  MoveL 667 to (47.33, 219.29, 110) mm, rotated rx -180 ry -65 rz 119.3 deg; joints [-3.014, -1.167, 27.755, -60.199, 92.729, -58.894, -1379.296]
  MoveL 668 to (51.17, 225.17, 120) mm, rotated rx 180 ry -65 rz 125.76 deg; joints [-2.739, -0.589, 26.527, -60.1, 93.267, -59.335, -1385.756]
  MoveL 669 to (54.3, 231.49, 130) mm, rotated rx 180 ry -65 rz 132.3 deg; joints [-2.464, 0.043, 25.187, -60.012, 93.835, -59.826, -1392.295]
  MoveL 670 to (56.65, 238.12, 140) mm, rotated rx -180 ry -65 rz 138.89 deg; joints [-2.19, 0.746, 23.7, -59.937, 94.442, -60.381, -1398.886]
  MoveL 671 to (58.18, 244.95, 150) mm, rotated rx -180 ry -65 rz 145.5 deg; joints [-1.917, 1.551, 22.008, -59.879, 95.103, -61.026, -1405.497]
  MoveL 672 to (58.89, 251.83, 160) mm, rotated rx -180 ry -65 rz 152.1 deg; joints [-1.644, 2.509, 20.004, -59.847, 95.845, -61.808, -1412.098]
  MoveL 673 to (58.8, 258.62, 170) mm, rotated rx -180 ry -65 rz 158.66 deg; joints [-1.372, 3.749, 17.431, -59.859, 96.733, -62.841, -1418.655]
  MoveL 674 to (57.96, 265.2, 180) mm, rotated rx 180 ry -65 rz 165.13 deg; joints [-1.101, 5.868, 13.081, -60.001, 98.071, -64.658, -1425.13]
  MoveL 675 to (55.81, 269.32, 189.23) mm, rotated rx -180 ry -65 rz 171.49 deg; joints [-0.831, 7.347, 10.028, -60.103, 99.08, -65.909, -1431.486]
  MoveL 676 to (53.44, 272.3, 198.22) mm, rotated rx -180 ry -65 rz 177.68 deg; joints [-0.562, 7.315, 10.028, -60.006, 99.318, -65.806, -1437.679]
  MoveL 677 to (51.74, 282.68, 210) mm, rotated rx -180 ry -65 rz 173.67 deg; joints [-0.015, -1.146, 27.158, -56.839, 99.081, -66.843, -1443.668]
  MoveL 678 to (48.8, 287.5, 220) mm, rotated rx -180 ry -65 rz 179.41 deg; joints [0.256, -0.417, 25.625, -56.812, 99.725, -67.39, -1449.406]
  MoveL 679 to (45.62, 291.76, 230) mm, rotated rx -180 ry -65 rz -175.15 deg; joints [0.525, 0.414, 23.888, -56.81, 100.426, -68.024, -1454.846]
  MoveL 680 to (42.34, 295.45, 240) mm, rotated rx -180 ry -65 rz -170.06 deg; joints [0.793, 1.393, 21.855, -56.845, 101.208, -68.785, -1459.941]
  MoveL 681 to (39.07, 298.58, 250) mm, rotated rx 180 ry -65 rz -165.36 deg; joints [1.06, 2.615, 19.337, -56.939, 102.123, -69.757, -1464.643]
  MoveL 682 to (35.92, 301.18, 260) mm, rotated rx -180 ry -65 rz -161.09 deg; joints [1.326, 4.38, 15.722, -57.163, 103.337, -71.21, -1468.905]
  MoveL 683 to (33.57, 302.05, 269.47) mm, rotated rx -180 ry -65 rz -157.32 deg; joints [1.591, 7.175, 10.028, -57.664, 105.11, -73.59, -1472.679]
  MoveL 684 to (32.63, 300.8, 278.13) mm, rotated rx 180 ry -65 rz -154.08 deg; joints [1.855, 7.155, 10.028, -57.554, 105.334, -73.468, -1475.919]
  MoveL 685 to (28.22, 306.19, 290) mm, rotated rx 180 ry -65 rz -161.42 deg; joints [2.42, 15.299, -6.738, -59.336, 114.508, -89.823, -1478.582]
  MoveL 686 to (-21.11, 309.47, 290) mm, rotated rx -180 ry -65 rz -106.89 deg; joints [2.421, 15.322, -6.805, -59.353, 114.532, -89.864, -1533.11]
  Set speed (60.0 mm/s)
  MoveL 687 to (-14.3, 309.76, 278.22) mm, rotated rx 180 ry -65 rz -99.58 deg; joints [1.857, 7.138, 10.028, -57.557, 105.344, -73.482, -1530.424]
  MoveL 688 to (-14.79, 311.04, 269.6) mm, rotated rx -180 ry -65 rz -102.86 deg; joints [1.594, 7.151, 10.028, -57.668, 105.125, -73.61, -1527.138]
  MoveL 689 to (-12.3, 312.09, 260) mm, rotated rx 180 ry -65 rz -106.71 deg; joints [1.33, 4.033, 16.354, -57.105, 103.186, -70.962, -1523.29]
  MoveL 690 to (-8.28, 312.8, 250) mm, rotated rx 180 ry -65 rz -111.08 deg; joints [1.065, 2.314, 19.855, -56.897, 102.008, -69.568, -1518.917]
  MoveL 691 to (-3.78, 313.26, 240) mm, rotated rx -180 ry -65 rz -115.94 deg; joints [0.799, 1.083, 22.369, -56.808, 101.101, -68.608, -1514.059]
  MoveL 692 to (1.16, 313.37, 230) mm, rotated rx 180 ry -65 rz -121.24 deg; joints [0.532, 0.083, 24.421, -56.775, 100.321, -67.848, -1508.756]
  MoveL 693 to (6.46, 313.03, 220) mm, rotated rx -180 ry -65 rz -126.95 deg; joints [0.264, -0.774, 26.185, -56.778, 99.621, -67.213, -1503.053]
  MoveL 694 to (12.04, 312.14, 210) mm, rotated rx -180 ry -65 rz -133.01 deg; joints [-0.005, -1.528, 27.745, -56.807, 98.976, -66.664, -1496.995]
  MoveL 695 to (20.33, 307.92, 198.7) mm, rotated rx -180 ry -65 rz -129.37 deg; joints [-0.551, 7.214, 10.028, -60.017, 99.377, -65.89, -1490.629]
  MoveL 696 to (24.04, 307.87, 189.76) mm, rotated rx -180 ry -65 rz -135.99 deg; joints [-0.82, 7.235, 10.028, -60.114, 99.145, -66.001, -1484.006]
  MoveL 697 to (29.38, 305.54, 180) mm, rotated rx -180 ry -65 rz -142.82 deg; joints [-1.089, 4.255, 16.095, -59.831, 97.379, -63.429, -1477.176]
  MoveL 698 to (34.94, 301.92, 170) mm, rotated rx 180 ry -65 rz -149.81 deg; joints [-1.359, 2.744, 19.201, -59.778, 96.359, -62.169, -1470.188]
  MoveL 699 to (40.17, 297.58, 160) mm, rotated rx 180 ry -65 rz -156.91 deg; joints [-1.631, 1.662, 21.443, -59.79, 95.559, -61.288, -1463.094]
  MoveL 700 to (44.94, 292.58, 150) mm, rotated rx -180 ry -65 rz -164.06 deg; joints [-1.903, 0.787, 23.27, -59.836, 94.864, -60.588, -1455.941]
  MoveL 701 to (49.15, 286.99, 140) mm, rotated rx -180 ry -65 rz -171.23 deg; joints [-2.176, 0.041, 24.838, -59.902, 94.236, -59.999, -1448.774]
  MoveL 702 to (52.68, 280.9, 130) mm, rotated rx -180 ry -65 rz -178.36 deg; joints [-2.45, -0.613, 26.225, -59.984, 93.655, -59.488, -1441.638]
  MoveL 703 to (55.46, 274.42, 120) mm, rotated rx 180 ry -65 rz 174.57 deg; joints [-2.726, -1.199, 27.475, -60.078, 93.108, -59.035, -1434.572]
  MoveL 704 to (55.84, 263.25, 108.59) mm, rotated rx 180 ry -65 rz 177.61 deg; joints [-3.24, 7.248, 10.028, -62.938, 93.374, -58.249, -1427.613]
  MoveL 705 to (57.58, 258.78, 99.33) mm, rotated rx 180 ry -65 rz 170.79 deg; joints [-3.514, 7.28, 10.028, -63.024, 93.127, -58.339, -1420.794]
  MoveL 706 to (58.95, 253.96, 90) mm, rotated rx -180 ry -65 rz 164.15 deg; joints [-3.787, 8.027, 8.582, -63.145, 93.209, -59.081, -1414.147]
  MoveL 707 to (58.51, 247.24, 80) mm, rotated rx 180 ry -65 rz 157.7 deg; joints [-4.062, 10.496, 3.656, -63.366, 94.079, -61.4, -1407.701]
  MoveL 708 to (57.35, 240.79, 70) mm, rotated rx -180 ry -65 rz 151.48 deg; joints [-4.337, 11.761, 1.161, -63.52, 94.39, -62.623, -1401.482]
  MoveL 709 to (55.55, 234.7, 60) mm, rotated rx -180 ry -65 rz 145.52 deg; joints [-4.613, 12.736, -0.752, -63.655, 94.566, -63.585, -1395.517]
  MoveL 710 to (53.21, 229.07, 50) mm, rotated rx -180 ry -65 rz 139.83 deg; joints [-4.889, 13.558, -2.357, -63.777, 94.67, -64.411, -1389.83]
  MoveL 711 to (50.45, 223.94, 40) mm, rotated rx 180 ry -65 rz 134.45 deg; joints [-5.166, 14.279, -3.764, -63.889, 94.728, -65.148, -1384.447]
  MoveL 712 to (47.39, 219.37, 30) mm, rotated rx 180 ry -65 rz 129.39 deg; joints [-5.444, 14.929, -5.029, -63.994, 94.753, -65.823, -1379.391]
  MoveL 713 to (44.15, 215.37, 20) mm, rotated rx 180 ry -65 rz 124.69 deg; joints [-5.721, 15.523, -6.184, -64.093, 94.753, -66.45, -1374.688]
  MoveL 714 to (40.85, 211.93, 10) mm, rotated rx -180 ry -65 rz 120.36 deg; joints [-6, 16.071, -7.253, -64.186, 94.732, -67.04, -1370.363]
  MoveL 715 to (33.26, 208.35, -1.05) mm, rotated rx 180 ry -65 rz 126.44 deg; joints [-6.466, 7.153, 10.028, -66.357, 87.195, -50.6, -1366.442]
  MoveL 716 to (-21.11, 309.47, 290) mm, rotated rx -180 ry -65 rz -106.89 deg; joints [2.421, 15.322, -6.805, -59.353, 114.532, -89.864, -1533.11]
  Set speed (60.0 mm/s)
  MoveL 717 to (-34.79, 325.15, 290) mm, rotated rx -180 ry -65 rz -101.9 deg; joints [2.347, 13.614, -2.112, -58.26, 112.923, -87.117, -1538.101]
  MoveL 718 to (33.26, 208.35, -1.05) mm, rotated rx -180 ry -65 rz 126.44 deg; joints [-6.466, 7.153, 10.028, -66.357, 87.195, -50.6, -1366.442]
  Set speed (60.0 mm/s)
  MoveL 719 to (55.59, 198.58, 0) mm, rotated rx 180 ry -65 rz 122.15 deg; joints [-6.324, 15.031, -3.912, -64.104, 93.441, -65.104, -1372.15]
  MoveL 720 to (33.26, 208.35, -1.05) mm, rotated rx -180 ry -65 rz 126.44 deg; joints [-6.466, 7.153, 10.028, -66.357, 87.195, -50.6, -1366.442]
  Set speed (60.0 mm/s)
  MoveL 721 to (40.85, 211.93, 10) mm, rotated rx -180 ry -65 rz 120.36 deg; joints [-6, 16.071, -7.253, -64.186, 94.732, -67.04, -1370.363]
  MoveL 722 to (44.15, 215.37, 20) mm, rotated rx 180 ry -65 rz 124.69 deg; joints [-5.721, 15.523, -6.184, -64.093, 94.753, -66.45, -1374.688]
  MoveL 723 to (47.39, 219.37, 30) mm, rotated rx 180 ry -65 rz 129.39 deg; joints [-5.444, 14.929, -5.029, -63.994, 94.753, -65.823, -1379.391]
  MoveL 724 to (50.45, 223.94, 40) mm, rotated rx 180 ry -65 rz 134.45 deg; joints [-5.166, 14.279, -3.764, -63.889, 94.728, -65.148, -1384.447]
  MoveL 725 to (53.21, 229.07, 50) mm, rotated rx -180 ry -65 rz 139.83 deg; joints [-4.889, 13.558, -2.357, -63.777, 94.67, -64.411, -1389.83]
  MoveL 726 to (55.55, 234.7, 60) mm, rotated rx 180 ry -65 rz 145.52 deg; joints [-4.613, 12.736, -0.752, -63.655, 94.566, -63.585, -1395.517]
  MoveL 727 to (57.35, 240.79, 70) mm, rotated rx -180 ry -65 rz 151.48 deg; joints [-4.337, 11.761, 1.161, -63.52, 94.39, -62.623, -1401.482]
  MoveL 728 to (58.51, 247.24, 80) mm, rotated rx 180 ry -65 rz 157.7 deg; joints [-4.062, 10.496, 3.656, -63.366, 94.079, -61.4, -1407.701]
  MoveL 729 to (58.95, 253.96, 90) mm, rotated rx 180 ry -65 rz 164.15 deg; joints [-3.787, 8.027, 8.582, -63.145, 93.209, -59.081, -1414.147]
  MoveL 730 to (57.58, 258.78, 99.33) mm, rotated rx -180 ry -65 rz 170.79 deg; joints [-3.514, 7.28, 10.028, -63.024, 93.127, -58.339, -1420.794]
  MoveL 731 to (55.84, 263.25, 108.59) mm, rotated rx 180 ry -65 rz 177.61 deg; joints [-3.24, 7.248, 10.028, -62.938, 93.374, -58.249, -1427.613]
  MoveL 732 to (55.46, 274.42, 120) mm, rotated rx -180 ry -65 rz 174.57 deg; joints [-2.726, 16.068, -7.419, -62.097, 101.684, -74.582, -1434.572]
  MoveL 733 to (52.68, 280.9, 130) mm, rotated rx 180 ry -65 rz -178.36 deg; joints [-2.45, 15.417, -6.169, -61.918, 101.643, -73.911, -1441.638]
  MoveL 734 to (49.15, 286.99, 140) mm, rotated rx -180 ry -65 rz -171.23 deg; joints [-2.176, 14.699, -4.782, -61.726, 101.566, -73.179, -1448.774]
  MoveL 735 to (44.94, 292.58, 150) mm, rotated rx -180 ry -65 rz -164.06 deg; joints [-1.903, 13.892, -3.214, -61.514, 101.44, -72.365, -1455.941]
  MoveL 736 to (40.17, 297.58, 160) mm, rotated rx -180 ry -65 rz -156.91 deg; joints [-1.631, 12.959, -1.387, -61.279, 101.247, -71.434, -1463.094]
  MoveL 737 to (34.94, 301.92, 170) mm, rotated rx -180 ry -65 rz -149.81 deg; joints [-1.359, 11.822, 0.855, -61.007, 100.945, -70.317, -1470.188]
  MoveL 738 to (29.38, 305.54, 180) mm, rotated rx -180 ry -65 rz -142.82 deg; joints [-1.089, 10.261, 3.96, -60.665, 100.423, -68.815, -1477.176]
  MoveL 739 to (24.04, 307.87, 189.76) mm, rotated rx 180 ry -65 rz -135.99 deg; joints [-0.82, 7.235, 10.028, -60.114, 99.145, -66.001, -1484.006]
  MoveL 740 to (20.33, 307.92, 198.7) mm, rotated rx -180 ry -65 rz -129.37 deg; joints [-0.551, 7.214, 10.028, -60.017, 99.377, -65.89, -1490.629]
  MoveL 741 to (12.04, 312.14, 210) mm, rotated rx 180 ry -65 rz -133.01 deg; joints [-0.005, -1.528, 27.745, -56.807, 98.976, -66.664, -1496.995]
  MoveL 742 to (6.46, 313.03, 220) mm, rotated rx 180 ry -65 rz -126.95 deg; joints [0.264, -0.774, 26.185, -56.778, 99.621, -67.213, -1503.053]
  MoveL 743 to (1.16, 313.37, 230) mm, rotated rx 180 ry -65 rz -121.24 deg; joints [0.532, 0.083, 24.421, -56.775, 100.321, -67.848, -1508.756]
  MoveL 744 to (-3.78, 313.26, 240) mm, rotated rx 180 ry -65 rz -115.94 deg; joints [0.799, 1.083, 22.369, -56.808, 101.101, -68.608, -1514.059]
  MoveL 745 to (-8.28, 312.8, 250) mm, rotated rx -180 ry -65 rz -111.08 deg; joints [1.065, 2.314, 19.855, -56.897, 102.008, -69.568, -1518.917]
  MoveL 746 to (-12.3, 312.09, 260) mm, rotated rx 180 ry -65 rz -106.71 deg; joints [1.33, 4.033, 16.354, -57.105, 103.186, -70.962, -1523.29]
  MoveL 747 to (-14.79, 311.04, 269.6) mm, rotated rx -180 ry -65 rz -102.86 deg; joints [1.594, 7.151, 10.028, -57.668, 105.125, -73.61, -1527.138]
  MoveL 748 to (-14.3, 309.76, 278.22) mm, rotated rx -180 ry -65 rz -99.58 deg; joints [1.857, 7.138, 10.028, -57.557, 105.344, -73.482, -1530.424]
  MoveL 749 to (-21.11, 309.47, 290) mm, rotated rx 180 ry -65 rz -106.89 deg; joints [2.421, -1.338, 26.861, -54.18, 105.153, -74.752, -1533.11]
  MoveL 750 to (-34.79, 325.15, 290) mm, rotated rx -180 ry -65 rz -101.9 deg; joints [2.347, 1.599, 22.168, -54.622, 106.121, -76.277, -1538.101]
  Set speed (60.0 mm/s)
  MoveL 751 to (-31.73, 326.57, 280) mm, rotated rx -180 ry -65 rz -104.51 deg; joints [2.083, 0.505, 24.407, -54.508, 105.261, -75.453, -1535.486]
  MoveL 752 to (-27.92, 328.13, 270) mm, rotated rx 180 ry -65 rz -107.71 deg; joints [1.818, -0.43, 26.324, -54.446, 104.496, -74.77, -1532.288]
  MoveL 753 to (-17.68, 328.71, 257.77) mm, rotated rx 180 ry -65 rz -101.46 deg; joints [1.26, 7.769, 10.028, -57.675, 104.526, -73.246, -1528.542]
  MoveL 754 to (-15.78, 330.54, 249.09) mm, rotated rx -180 ry -65 rz -105.71 deg; joints [0.996, 7.782, 10.028, -57.788, 104.306, -73.373, -1524.286]
  MoveL 755 to (-12.17, 332.29, 240) mm, rotated rx -180 ry -65 rz -110.44 deg; joints [0.731, 5.846, 13.967, -57.494, 103.022, -71.769, -1519.557]
  MoveL 756 to (-5.61, 333.04, 230) mm, rotated rx -180 ry -65 rz -115.61 deg; joints [0.465, 3.66, 18.415, -57.203, 101.592, -69.958, -1514.392]
  MoveL 757 to (1.49, 333.22, 220) mm, rotated rx -180 ry -65 rz -121.17 deg; joints [0.198, 2.31, 21.174, -57.1, 100.621, -68.887, -1508.834]
  MoveL 758 to (9.03, 332.72, 210) mm, rotated rx -180 ry -65 rz -127.08 deg; joints [-0.071, 1.257, 23.337, -57.066, 99.812, -68.076, -1502.922]
  MoveL 759 to (16.88, 331.41, 200) mm, rotated rx -180 ry -65 rz -133.3 deg; joints [-0.34, 0.375, 25.158, -57.071, 99.097, -67.411, -1496.702]
  MoveL 760 to (24.89, 329.2, 190) mm, rotated rx -180 ry -65 rz -139.78 deg; joints [-0.61, -0.391, 26.749, -57.103, 98.444, -66.845, -1490.217]
  MoveL 761 to (36.37, 321.13, 177.97) mm, rotated rx 180 ry -65 rz -136.49 deg; joints [-1.15, 7.85, 10.028, -60.155, 98.565, -65.62, -1483.513]
  MoveL 762 to (42.24, 319.12, 168.96) mm, rotated rx -180 ry -65 rz -143.36 deg; joints [-1.42, 7.875, 10.028, -60.254, 98.331, -65.728, -1476.637]
  MoveL 763 to (48.36, 316.44, 159.89) mm, rotated rx -180 ry -65 rz -150.37 deg; joints [-1.69, 7.901, 10.028, -60.352, 98.094, -65.833, -1469.635]
  MoveL 764 to (55.2, 310.67, 150) mm, rotated rx 180 ry -65 rz -157.45 deg; joints [-1.962, 11.044, 3.733, -60.871, 99.414, -68.741, -1462.551]
  MoveL 765 to (61.48, 303.74, 140) mm, rotated rx -180 ry -65 rz -164.57 deg; joints [-2.234, 12.483, 0.887, -61.168, 99.865, -70.12, -1455.431]
  MoveL 766 to (66.92, 296.06, 130) mm, rotated rx -180 ry -65 rz -171.68 deg; joints [-2.507, 13.555, -1.216, -61.411, 100.126, -71.168, -1448.317]
  MoveL 767 to (71.41, 287.77, 120) mm, rotated rx 180 ry -65 rz -178.75 deg; joints [-2.782, 14.443, -2.946, -61.624, 100.292, -72.05, -1441.249]
  MoveL 768 to (74.87, 279.04, 110) mm, rotated rx -180 ry -65 rz 174.27 deg; joints [-3.057, 15.216, -4.44, -61.816, 100.396, -72.826, -1434.266]
  MoveL 769 to (77.24, 270.04, 100) mm, rotated rx -180 ry -65 rz 167.4 deg; joints [-3.333, 15.907, -5.769, -61.993, 100.457, -73.527, -1427.404]
  MoveL 770 to (78.53, 260.95, 90) mm, rotated rx 180 ry -65 rz 160.7 deg; joints [-3.609, 16.536, -6.973, -62.158, 100.485, -74.174, -1420.696]
  MoveL 771 to (75.48, 247.1, 78.35) mm, rotated rx -180 ry -65 rz 164.17 deg; joints [-4.113, 7.925, 10.028, -63.191, 92.325, -58.021, -1414.174]
  MoveL 772 to (75.7, 240.53, 69.02) mm, rotated rx 180 ry -65 rz 157.87 deg; joints [-4.388, 7.956, 10.028, -63.279, 92.078, -58.111, -1407.868]
  MoveL 773 to (75.43, 234.04, 59.66) mm, rotated rx -180 ry -65 rz 151.81 deg; joints [-4.663, 7.986, 10.028, -63.367, 91.831, -58.202, -1401.808]
  MoveL 774 to (73.92, 227.12, 50) mm, rotated rx -180 ry -65 rz 146.02 deg; joints [-4.938, 6.02, 14.06, -63.419, 90.673, -56.471, -1396.021]
  MoveL 775 to (70.87, 219.96, 40) mm, rotated rx -180 ry -65 rz 140.54 deg; joints [-5.214, 4.454, 17.278, -63.513, 89.704, -55.108, -1390.535]
  MoveL 776 to (67.34, 213.5, 30) mm, rotated rx 180 ry -65 rz 135.38 deg; joints [-5.491, 3.412, 19.436, -63.628, 88.978, -54.223, -1385.378]
  MoveL 777 to (63.51, 207.78, 20) mm, rotated rx -180 ry -65 rz 130.58 deg; joints [-5.768, 2.578, 21.169, -63.754, 88.351, -53.53, -1380.576]
  MoveL 778 to (59.54, 202.81, 10) mm, rotated rx -180 ry -65 rz 126.16 deg; joints [-6.046, 1.865, 22.654, -63.887, 87.783, -52.949, -1376.157]
  MoveL 779 to (55.59, 198.58, 0) mm, rotated rx -180 ry -65 rz 122.15 deg; joints [-6.324, 1.235, 23.968, -64.026, 87.256, -52.444, -1372.15]
  MoveL 780 to (-34.79, 325.15, 290) mm, rotated rx 180 ry -65 rz -101.9 deg; joints [2.347, 1.599, 22.168, -54.622, 106.121, -76.277, -1538.101]
  Set speed (60.0 mm/s)
  MoveL 781 to (-30.72, 304.75, 290) mm, rotated rx 180 ry -65 rz -95.53 deg; joints [2.42, -1.275, 26.764, -54.188, 105.172, -74.782, -1544.467]
  MoveL 782 to (55.59, 198.58, 0) mm, rotated rx 180 ry -65 rz 122.15 deg; joints [-6.324, 1.235, 23.968, -64.026, 87.256, -52.444, -1372.15]
  Set speed (60.0 mm/s)
  MoveL 783 to (41.3, 215.27, -0.99) mm, rotated rx 180 ry -65 rz 136.17 deg; joints [-6.465, 7.133, 10.028, -66.356, 87.204, -50.617, -1376.169]
  MoveL 784 to (55.59, 198.58, 0) mm, rotated rx -180 ry -65 rz 122.15 deg; joints [-6.324, 1.235, 23.968, -64.026, 87.256, -52.444, -1372.15]
  Set speed (60.0 mm/s)
  MoveL 785 to (59.54, 202.81, 10) mm, rotated rx -180 ry -65 rz 126.16 deg; joints [-6.046, 1.865, 22.654, -63.887, 87.783, -52.949, -1376.157]
  MoveL 786 to (63.51, 207.78, 20) mm, rotated rx -180 ry -65 rz 130.58 deg; joints [-5.768, 2.578, 21.169, -63.754, 88.351, -53.53, -1380.576]
  MoveL 787 to (67.34, 213.5, 30) mm, rotated rx -180 ry -65 rz 135.38 deg; joints [-5.491, 3.412, 19.436, -63.628, 88.978, -54.223, -1385.378]
  MoveL 788 to (70.87, 219.96, 40) mm, rotated rx 180 ry -65 rz 140.54 deg; joints [-5.214, 4.454, 17.278, -63.513, 89.704, -55.108, -1390.535]
  MoveL 789 to (73.92, 227.12, 50) mm, rotated rx 180 ry -65 rz 146.02 deg; joints [-4.938, 6.02, 14.06, -63.419, 90.673, -56.471, -1396.021]
  MoveL 790 to (75.43, 234.04, 59.66) mm, rotated rx -180 ry -65 rz 151.81 deg; joints [-4.663, 7.986, 10.028, -63.367, 91.831, -58.202, -1401.808]
  MoveL 791 to (75.7, 240.53, 69.02) mm, rotated rx -180 ry -65 rz 157.87 deg; joints [-4.388, 7.956, 10.028, -63.279, 92.078, -58.111, -1407.868]
  MoveL 792 to (75.48, 247.1, 78.35) mm, rotated rx 180 ry -65 rz 164.17 deg; joints [-4.113, 7.925, 10.028, -63.191, 92.325, -58.021, -1414.174]
  MoveL 793 to (78.53, 260.95, 90) mm, rotated rx -180 ry -65 rz 160.7 deg; joints [-3.609, -0.289, 27.028, -60.472, 92.192, -59.025, -1420.696]
  MoveL 794 to (77.24, 270.04, 100) mm, rotated rx 180 ry -65 rz 167.4 deg; joints [-3.333, 0.273, 25.825, -60.367, 92.724, -59.461, -1427.404]
  MoveL 795 to (74.87, 279.04, 110) mm, rotated rx -180 ry -65 rz 174.27 deg; joints [-3.057, 0.897, 24.496, -60.273, 93.289, -59.951, -1434.266]
  MoveL 796 to (71.41, 287.77, 120) mm, rotated rx -180 ry -65 rz -178.75 deg; joints [-2.782, 1.603, 23.002, -60.192, 93.897, -60.513, -1441.249]
  MoveL 797 to (66.92, 296.06, 130) mm, rotated rx -180 ry -65 rz -171.68 deg; joints [-2.507, 2.427, 21.272, -60.129, 94.565, -61.176, -1448.317]
  MoveL 798 to (61.48, 303.74, 140) mm, rotated rx 180 ry -65 rz -164.57 deg; joints [-2.234, 3.436, 19.169, -60.093, 95.328, -62.003, -1455.431]
  MoveL 799 to (55.2, 310.67, 150) mm, rotated rx -180 ry -65 rz -157.45 deg; joints [-1.962, 4.814, 16.322, -60.108, 96.279, -63.155, -1462.551]
  MoveL 800 to (48.36, 316.44, 159.89) mm, rotated rx 180 ry -65 rz -150.37 deg; joints [-1.69, 7.901, 10.028, -60.352, 98.094, -65.833, -1469.635]
  MoveL 801 to (42.24, 319.12, 168.96) mm, rotated rx -180 ry -65 rz -143.36 deg; joints [-1.42, 7.875, 10.028, -60.254, 98.331, -65.728, -1476.637]
  MoveL 802 to (36.37, 321.13, 177.97) mm, rotated rx -180 ry -65 rz -136.49 deg; joints [-1.15, 7.85, 10.028, -60.155, 98.565, -65.62, -1483.513]
  MoveL 803 to (24.89, 329.2, 190) mm, rotated rx -180 ry -65 rz -139.78 deg; joints [-0.61, 16.157, -6.693, -60.422, 107.256, -81.648, -1490.217]
  MoveL 804 to (16.88, 331.41, 200) mm, rotated rx 180 ry -65 rz -133.3 deg; joints [-0.34, 15.349, -5.102, -60.125, 107.099, -80.798, -1496.702]
  MoveL 805 to (9.03, 332.72, 210) mm, rotated rx -180 ry -65 rz -127.08 deg; joints [-0.071, 14.429, -3.281, -59.796, 106.877, -79.844, -1502.922]
  MoveL 806 to (1.49, 333.22, 220) mm, rotated rx 180 ry -65 rz -121.17 deg; joints [0.198, 13.342, -1.118, -59.423, 106.559, -78.736, -1508.834]
  MoveL 807 to (-5.61, 333.04, 230) mm, rotated rx -180 ry -65 rz -115.61 deg; joints [0.465, 11.961, 1.641, -58.978, 106.077, -77.364, -1514.392]
  MoveL 808 to (-12.17, 332.29, 240) mm, rotated rx -180 ry -65 rz -110.44 deg; joints [0.731, 9.745, 6.088, -58.34, 105.136, -75.246, -1519.557]
  MoveL 809 to (-15.78, 330.54, 249.09) mm, rotated rx -180 ry -65 rz -105.71 deg; joints [0.996, 7.782, 10.028, -57.788, 104.306, -73.373, -1524.286]
  MoveL 810 to (-17.68, 328.71, 257.77) mm, rotated rx -180 ry -65 rz -101.46 deg; joints [1.26, 7.769, 10.028, -57.675, 104.526, -73.246, -1528.542]
  MoveL 811 to (-27.92, 328.13, 270) mm, rotated rx 180 ry -65 rz -107.71 deg; joints [1.818, 15.697, -6.268, -59.233, 113.553, -89.338, -1532.288]
  MoveL 812 to (-31.73, 326.57, 280) mm, rotated rx -180 ry -65 rz -104.51 deg; joints [2.083, 14.735, -4.351, -58.774, 113.285, -88.299, -1535.486]
  MoveL 813 to (-34.79, 325.15, 290) mm, rotated rx -180 ry -65 rz -101.9 deg; joints [2.347, 13.614, -2.112, -58.26, 112.923, -87.117, -1538.101]
  MoveL 814 to (-30.72, 304.75, 290) mm, rotated rx 180 ry -65 rz -95.53 deg; joints [2.42, 15.288, -6.708, -59.329, 114.498, -89.805, -1544.467]
  Set speed (60.0 mm/s)
  MoveL 815 to (-23.89, 306.35, 278.15) mm, rotated rx 180 ry -65 rz -88.19 deg; joints [1.855, 7.151, 10.028, -57.554, 105.336, -73.471, -1541.806]
  MoveL 816 to (-24.62, 307.45, 269.53) mm, rotated rx -180 ry -65 rz -91.45 deg; joints [1.592, 7.162, 10.028, -57.666, 105.118, -73.6, -1538.548]
  MoveL 817 to (-22.53, 308.91, 260) mm, rotated rx -180 ry -65 rz -95.27 deg; joints [1.329, 10.215, 3.881, -58.52, 106.538, -76.47, -1534.728]
  MoveL 818 to (-18.7, 310.34, 250) mm, rotated rx -180 ry -65 rz -99.62 deg; joints [1.064, 12.003, 0.29, -59.089, 107.252, -78.221, -1530.381]
  MoveL 819 to (-14.35, 311.61, 240) mm, rotated rx 180 ry -65 rz -104.46 deg; joints [0.799, 13.279, -2.266, -59.531, 107.681, -79.514, -1525.543]
  MoveL 820 to (-9.52, 312.61, 230) mm, rotated rx -180 ry -65 rz -109.75 deg; joints [0.532, 14.321, -4.347, -59.911, 107.979, -80.596, -1520.254]
  MoveL 821 to (-4.24, 313.23, 220) mm, rotated rx 180 ry -65 rz -115.45 deg; joints [0.265, 15.218, -6.134, -60.25, 108.194, -81.546, -1514.554]
  MoveL 822 to (1.41, 313.37, 210) mm, rotated rx 180 ry -65 rz -121.51 deg; joints [-0.004, 16.014, -7.714, -60.559, 108.35, -82.402, -1508.487]
  MoveL 823 to (10.28, 310.83, 198.74) mm, rotated rx -180 ry -65 rz -117.9 deg; joints [-0.551, 7.207, 10.028, -60.017, 99.382, -65.896, -1502.098]
  MoveL 824 to (13.88, 311.45, 189.81) mm, rotated rx -180 ry -65 rz -124.57 deg; joints [-0.818, 7.224, 10.028, -60.115, 99.151, -66.01, -1495.435]
  MoveL 825 to (19.65, 310.01, 180) mm, rotated rx -180 ry -65 rz -131.45 deg; joints [-1.087, 4.115, 16.351, -59.818, 97.322, -63.328, -1488.548]
  MoveL 826 to (25.78, 307.45, 170) mm, rotated rx 180 ry -65 rz -138.51 deg; joints [-1.357, 2.623, 19.411, -59.769, 96.316, -62.091, -1481.489]
  MoveL 827 to (31.7, 304.13, 160) mm, rotated rx 180 ry -65 rz -145.69 deg; joints [-1.628, 1.542, 21.643, -59.783, 95.52, -61.217, -1474.307]
  MoveL 828 to (37.3, 300.08, 150) mm, rotated rx -180 ry -65 rz -152.95 deg; joints [-1.901, 0.666, 23.467, -59.829, 94.828, -60.521, -1467.054]
  MoveL 829 to (42.45, 295.34, 140) mm, rotated rx 180 ry -65 rz -160.22 deg; joints [-2.174, -0.08, 25.033, -59.896, 94.202, -59.935, -1459.778]
  MoveL 830 to (47.02, 289.99, 130) mm, rotated rx 180 ry -65 rz -167.48 deg; joints [-2.448, -0.735, 26.417, -59.979, 93.622, -59.427, -1452.524]
  MoveL 831 to (50.93, 284.12, 120) mm, rotated rx -180 ry -65 rz -174.66 deg; joints [-2.723, -1.321, 27.664, -60.073, 93.077, -58.977, -1445.337]
  MoveL 832 to (53.41, 273.61, 108.72) mm, rotated rx -180 ry -65 rz -171.74 deg; joints [-3.238, 7.218, 10.028, -62.939, 93.39, -58.274, -1438.256]
  MoveL 833 to (55.97, 269.53, 99.46) mm, rotated rx -180 ry -65 rz -178.68 deg; joints [-3.511, 7.25, 10.028, -63.025, 93.143, -58.365, -1431.316]
  MoveL 834 to (58.06, 264.62, 90) mm, rotated rx -180 ry -65 rz 174.55 deg; joints [-3.785, 8.775, 7.009, -63.188, 93.584, -59.818, -1424.553]
  MoveL 835 to (58.85, 257.94, 80) mm, rotated rx 180 ry -65 rz 168 deg; joints [-4.059, 10.726, 3.129, -63.384, 94.214, -61.664, -1417.997]
  MoveL 836 to (58.87, 251.39, 70) mm, rotated rx -180 ry -65 rz 161.68 deg; joints [-4.335, 11.918, 0.782, -63.535, 94.491, -62.821, -1411.675]
  MoveL 837 to (58.2, 245.07, 60) mm, rotated rx -180 ry -65 rz 155.62 deg; joints [-4.61, 12.858, -1.057, -63.668, 94.649, -63.749, -1405.616]
  MoveL 838 to (56.92, 239.11, 50) mm, rotated rx 180 ry -65 rz 149.84 deg; joints [-4.887, 13.657, -2.614, -63.788, 94.742, -64.551, -1399.845]
  MoveL 839 to (55.13, 233.57, 40) mm, rotated rx 180 ry -65 rz 144.39 deg; joints [-5.164, 14.362, -3.984, -63.899, 94.791, -65.271, -1394.385]
  MoveL 840 to (52.95, 228.52, 30) mm, rotated rx -180 ry -65 rz 139.26 deg; joints [-5.442, 14.998, -5.22, -64.003, 94.808, -65.932, -1389.263]
  MoveL 841 to (50.48, 223.99, 20) mm, rotated rx 180 ry -65 rz 134.5 deg; joints [-5.72, 15.582, -6.351, -64.101, 94.802, -66.547, -1384.503]
  MoveL 842 to (42.09, 217.59, 8.47) mm, rotated rx -180 ry -65 rz 140.13 deg; joints [-6.189, 7.114, 10.028, -66.279, 87.453, -50.529, -1380.13]
  MoveL 843 to (41.3, 215.27, -0.99) mm, rotated rx 180 ry -65 rz 136.17 deg; joints [-6.465, 7.133, 10.028, -66.356, 87.204, -50.617, -1376.169]
  MoveL 844 to (-30.72, 304.75, 290) mm, rotated rx -180 ry -65 rz -95.53 deg; joints [2.42, 15.288, -6.708, -59.329, 114.498, -89.805, -1544.467]
  Set speed (60.0 mm/s)
  MoveL 845 to (-58.22, 263.67, 290) mm, rotated rx -180 ry -65 rz -43.61 deg; joints [2.405, 14.999, -5.871, -59.121, 114.205, -89.297, -1596.394]
  MoveL 846 to (41.3, 215.27, -0.99) mm, rotated rx 180 ry -65 rz 136.17 deg; joints [-6.465, 7.133, 10.028, -66.356, 87.204, -50.617, -1736.169]
  Set speed (60.0 mm/s)
  MoveL 847 to (57.25, 262.28, -0.53) mm, rotated rx -180 ry -65 rz -175.75 deg; joints [-6.455, 7, 10.028, -66.348, 87.266, -50.736, -1784.254]
  MoveL 848 to (41.3, 215.27, -0.99) mm, rotated rx -180 ry -65 rz 136.17 deg; joints [-6.465, 7.133, 10.028, -66.356, 87.204, -50.617, -1736.169]
  Set speed (60.0 mm/s)
  MoveL 849 to (42.09, 217.59, 8.47) mm, rotated rx -180 ry -65 rz 140.13 deg; joints [-6.189, 7.114, 10.028, -66.279, 87.453, -50.529, -1740.13]
  MoveL 850 to (50.48, 223.99, 20) mm, rotated rx -180 ry -65 rz 134.5 deg; joints [-5.72, -0.628, 26.407, -63.801, 87.493, -51.686, -1744.503]
  MoveL 851 to (52.95, 228.52, 30) mm, rotated rx 180 ry -65 rz 139.26 deg; joints [-5.442, -0.092, 25.275, -63.664, 87.982, -52.109, -1749.263]
  MoveL 852 to (55.13, 233.57, 40) mm, rotated rx -180 ry -65 rz 144.39 deg; joints [-5.164, 0.494, 24.04, -63.533, 88.496, -52.579, -1754.385]
  MoveL 853 to (56.92, 239.11, 50) mm, rotated rx -180 ry -65 rz 149.84 deg; joints [-4.887, 1.145, 22.67, -63.408, 89.044, -53.11, -1759.845]
  MoveL 854 to (58.2, 245.07, 60) mm, rotated rx -180 ry -65 rz 155.62 deg; joints [-4.61, 1.887, 21.113, -63.291, 89.636, -53.725, -1765.616]
  MoveL 855 to (58.87, 251.39, 70) mm, rotated rx 180 ry -65 rz 161.68 deg; joints [-4.335, 2.768, 19.274, -63.185, 90.295, -54.466, -1771.675]
  MoveL 856 to (58.85, 257.94, 80) mm, rotated rx -180 ry -65 rz 168 deg; joints [-4.059, 3.899, 16.926, -63.096, 91.073, -55.435, -1777.997]
  MoveL 857 to (58.06, 264.62, 90) mm, rotated rx 180 ry -65 rz 174.55 deg; joints [-3.785, 5.787, 13.046, -63.051, 92.205, -57.094, -1784.553]
  MoveL 858 to (55.97, 269.53, 99.46) mm, rotated rx 180 ry -65 rz -178.68 deg; joints [-3.511, 7.25, 10.028, -63.025, 93.143, -58.365, -1791.316]
  MoveL 859 to (53.41, 273.61, 108.72) mm, rotated rx -180 ry -65 rz -171.74 deg; joints [-3.238, 7.218, 10.028, -62.939, 93.39, -58.274, -1798.256]
  MoveL 860 to (50.93, 284.12, 120) mm, rotated rx -180 ry -65 rz -174.66 deg; joints [-2.723, 16.132, -7.608, -62.119, 101.745, -74.693, -1805.337]
  MoveL 861 to (47.02, 289.99, 130) mm, rotated rx 180 ry -65 rz -167.48 deg; joints [-2.448, 15.484, -6.361, -61.941, 101.704, -74.022, -1812.524]
  MoveL 862 to (42.45, 295.34, 140) mm, rotated rx 180 ry -65 rz -160.22 deg; joints [-2.174, 14.769, -4.977, -61.747, 101.626, -73.289, -1819.778]
  MoveL 863 to (37.3, 300.08, 150) mm, rotated rx -180 ry -65 rz -152.95 deg; joints [-1.901, 13.966, -3.411, -61.535, 101.5, -72.474, -1827.054]
  MoveL 864 to (31.7, 304.13, 160) mm, rotated rx 180 ry -65 rz -145.69 deg; joints [-1.628, 13.038, -1.587, -61.299, 101.307, -71.542, -1834.307]
  MoveL 865 to (25.78, 307.45, 170) mm, rotated rx 180 ry -65 rz -138.51 deg; joints [-1.357, 11.909, 0.645, -61.027, 101.007, -70.426, -1841.489]
  MoveL 866 to (19.65, 310.01, 180) mm, rotated rx 180 ry -65 rz -131.45 deg; joints [-1.087, 10.373, 3.705, -60.688, 100.494, -68.941, -1848.548]
  MoveL 867 to (13.88, 311.45, 189.81) mm, rotated rx -180 ry -65 rz -124.57 deg; joints [-0.818, 7.224, 10.028, -60.115, 99.151, -66.01, -1855.435]
  MoveL 868 to (10.28, 310.83, 198.74) mm, rotated rx 180 ry -65 rz -117.9 deg; joints [-0.551, 7.207, 10.028, -60.017, 99.382, -65.896, -1862.098]
  MoveL 869 to (1.41, 313.37, 210) mm, rotated rx -180 ry -65 rz -121.51 deg; joints [-0.004, -1.544, 27.77, -56.806, 98.972, -66.657, -1868.487]
  MoveL 870 to (-4.24, 313.23, 220) mm, rotated rx -180 ry -65 rz -115.45 deg; joints [0.265, -0.777, 26.19, -56.778, 99.62, -67.212, -1874.554]
  MoveL 871 to (-9.52, 312.61, 230) mm, rotated rx 180 ry -65 rz -109.75 deg; joints [0.532, 0.094, 24.402, -56.777, 100.325, -67.855, -1880.254]
  MoveL 872 to (-14.35, 311.61, 240) mm, rotated rx -180 ry -65 rz -104.46 deg; joints [0.799, 1.112, 22.322, -56.811, 101.111, -68.624, -1885.543]
  MoveL 873 to (-18.7, 310.34, 250) mm, rotated rx -180 ry -65 rz -99.62 deg; joints [1.064, 2.365, 19.766, -56.904, 102.028, -69.601, -1890.381]
  MoveL 874 to (-22.53, 308.91, 260) mm, rotated rx -180 ry -65 rz -95.27 deg; joints [1.329, 4.131, 16.175, -57.122, 103.228, -71.032, -1894.728]
  MoveL 875 to (-24.62, 307.45, 269.53) mm, rotated rx 180 ry -65 rz -91.45 deg; joints [1.592, 7.162, 10.028, -57.666, 105.118, -73.6, -1898.548]
  MoveL 876 to (-23.89, 306.35, 278.15) mm, rotated rx 180 ry -65 rz -88.19 deg; joints [1.855, 7.151, 10.028, -57.554, 105.336, -73.471, -1901.806]
  MoveL 877 to (-30.72, 304.75, 290) mm, rotated rx -180 ry -65 rz -95.53 deg; joints [2.42, -1.275, 26.764, -54.188, 105.172, -74.782, -1904.467]
  MoveL 878 to (-58.22, 263.67, 290) mm, rotated rx -180 ry -65 rz -43.61 deg; joints [2.405, -0.736, 25.927, -54.263, 105.335, -75.041, -1956.394]
  Set speed (60.0 mm/s)
  MoveL 879 to (-57.77, 266.15, 280) mm, rotated rx -180 ry -65 rz -46.08 deg; joints [2.141, -1.618, 27.728, -54.215, 104.605, -74.413, -1953.924]
  MoveL 880 to (-55.45, 271.33, 268.93) mm, rotated rx 180 ry -65 rz -39.11 deg; joints [1.579, 7.278, 10.028, -57.645, 105.045, -73.506, -1950.894]
  MoveL 881 to (-56.08, 272.6, 260) mm, rotated rx -180 ry -65 rz -42.67 deg; joints [1.316, 5.488, 13.657, -57.363, 103.847, -72.043, -1947.333]
  MoveL 882 to (-54.69, 276.44, 250) mm, rotated rx -180 ry -65 rz -46.73 deg; joints [1.052, 3.098, 18.494, -57.008, 102.312, -70.069, -1943.267]
  MoveL 883 to (-52.84, 280.57, 240) mm, rotated rx 180 ry -65 rz -51.28 deg; joints [0.788, 1.654, 21.421, -56.876, 101.299, -68.937, -1938.724]
  MoveL 884 to (-50.46, 284.91, 230) mm, rotated rx 180 ry -65 rz -56.27 deg; joints [0.523, 0.519, 23.719, -56.821, 100.459, -68.08, -1933.731]
  MoveL 885 to (-47.51, 289.33, 220) mm, rotated rx -180 ry -65 rz -61.68 deg; joints [0.256, -0.443, 25.665, -56.81, 99.718, -67.377, -1928.316]
  MoveL 886 to (-43.95, 293.72, 210) mm, rotated rx 180 ry -65 rz -67.49 deg; joints [-0.011, -1.288, 27.377, -56.827, 99.042, -66.776, -1922.509]
  MoveL 887 to (-35.74, 299.31, 198.51) mm, rotated rx -180 ry -65 rz -63.66 deg; joints [-0.556, 7.253, 10.028, -60.012, 99.354, -65.858, -1916.342]
  MoveL 888 to (-34, 302.1, 189.66) mm, rotated rx -180 ry -65 rz -70.15 deg; joints [-0.822, 7.255, 10.028, -60.112, 99.133, -65.984, -1909.847]
  MoveL 889 to (-29.57, 305.43, 180) mm, rotated rx -180 ry -65 rz -76.94 deg; joints [-1.089, 10.258, 3.967, -60.665, 100.421, -68.812, -1903.063]
  MoveL 890 to (-23.65, 308.43, 170) mm, rotated rx 180 ry -65 rz -83.97 deg; joints [-1.357, 11.924, 0.608, -61.031, 101.018, -70.445, -1896.03]
  MoveL 891 to (-17.28, 310.79, 160) mm, rotated rx 180 ry -65 rz -91.21 deg; joints [-1.626, 13.117, -1.789, -61.32, 101.368, -71.651, -1888.791]
  MoveL 892 to (-10.57, 312.43, 150) mm, rotated rx 180 ry -65 rz -98.61 deg; joints [-1.897, 14.087, -3.734, -61.571, 101.6, -72.653, -1881.395]
  MoveL 893 to (-3.62, 313.27, 140) mm, rotated rx 180 ry -65 rz -106.11 deg; joints [-2.168, 14.92, -5.395, -61.795, 101.758, -73.528, -1873.889]
  MoveL 894 to (3.42, 313.28, 130) mm, rotated rx -180 ry -65 rz -113.67 deg; joints [-2.441, 15.657, -6.857, -61.998, 101.862, -74.311, -1866.327]
  MoveL 895 to (14.77, 308.97, 118.31) mm, rotated rx -180 ry -65 rz -111.24 deg; joints [-2.957, 7.1, 10.028, -62.855, 93.682, -58.257, -1858.761]
  MoveL 896 to (19.25, 308.72, 109.14) mm, rotated rx -180 ry -65 rz -118.76 deg; joints [-3.228, 7.118, 10.028, -62.941, 93.443, -58.36, -1851.243]
  MoveL 897 to (23.94, 308.16, 99.92) mm, rotated rx -180 ry -65 rz -126.18 deg; joints [-3.501, 7.137, 10.028, -63.027, 93.203, -58.46, -1843.825]
  MoveL 898 to (29.89, 305.25, 90) mm, rotated rx 180 ry -65 rz -133.45 deg; joints [-3.774, 4.15, 16.109, -63.005, 91.568, -55.819, -1836.554]
  MoveL 899 to (35.48, 301.51, 80) mm, rotated rx -180 ry -65 rz -140.52 deg; joints [-4.048, 2.832, 18.819, -63.081, 90.709, -54.694, -1829.477]
  MoveL 900 to (40.49, 297.28, 70) mm, rotated rx -180 ry -65 rz -147.36 deg; joints [-4.323, 1.865, 20.824, -63.179, 90.013, -53.883, -1822.636]
  MoveL 901 to (44.86, 292.68, 60) mm, rotated rx -180 ry -65 rz -153.93 deg; joints [-4.599, 1.074, 22.473, -63.291, 89.399, -53.23, -1816.069]
  MoveL 902 to (48.58, 287.83, 50) mm, rotated rx -180 ry -65 rz -160.19 deg; joints [-4.875, 0.396, 23.898, -63.412, 88.839, -52.677, -1809.813]
  MoveL 903 to (51.63, 282.88, 40) mm, rotated rx 180 ry -65 rz -166.1 deg; joints [-5.152, -0.204, 25.163, -63.539, 88.316, -52.194, -1803.9]
  MoveL 904 to (54.06, 277.94, 30) mm, rotated rx -180 ry -65 rz -171.64 deg; joints [-5.43, -0.746, 26.31, -63.672, 87.822, -51.763, -1798.36]
  MoveL 905 to (55.91, 273.13, 20) mm, rotated rx 180 ry -65 rz -176.78 deg; joints [-5.709, -1.242, 27.364, -63.81, 87.351, -51.373, -1793.221]
  MoveL 906 to (55.85, 264.47, 8.94) mm, rotated rx -180 ry -65 rz -171.49 deg; joints [-6.179, 6.978, 10.028, -66.271, 87.517, -50.65, -1788.51]
  MoveL 907 to (57.25, 262.28, -0.53) mm, rotated rx 180 ry -65 rz -175.75 deg; joints [-6.455, 7, 10.028, -66.348, 87.266, -50.736, -1784.254]
  MoveL 908 to (-58.22, 263.67, 290) mm, rotated rx -180 ry -65 rz -43.61 deg; joints [2.405, 14.999, -5.871, -59.121, 114.205, -89.297, -1956.394]
  Set speed (60.0 mm/s)
  MoveL 909 to (-78.63, 259.66, 290) mm, rotated rx -180 ry -65 rz -39.75 deg; joints [2.329, 13.048, -0.675, -57.958, 112.448, -86.325, -1960.245]
  MoveL 910 to (57.25, 262.28, -0.53) mm, rotated rx 180 ry -65 rz -175.75 deg; joints [-6.455, 7, 10.028, -66.348, 87.266, -50.736, -1784.254]
  Set speed (60.0 mm/s)
  MoveL 911 to (76.17, 274.65, 0) mm, rotated rx -180 ry -65 rz -179.11 deg; joints [-6.312, 0.429, 25.273, -64.043, 87.048, -51.99, -1790.889]
  MoveL 912 to (57.25, 262.28, -0.53) mm, rotated rx -180 ry -65 rz -175.75 deg; joints [-6.455, 7, 10.028, -66.348, 87.266, -50.736, -1784.254]
  Set speed (60.0 mm/s)
  MoveL 913 to (55.85, 264.47, 8.94) mm, rotated rx 180 ry -65 rz -171.49 deg; joints [-6.179, 6.978, 10.028, -66.271, 87.517, -50.65, -1788.51]
  MoveL 914 to (55.91, 273.13, 20) mm, rotated rx -180 ry -65 rz -176.78 deg; joints [-5.709, -1.242, 27.364, -63.81, 87.351, -51.373, -1793.221]
  MoveL 915 to (54.06, 277.94, 30) mm, rotated rx 180 ry -65 rz -171.64 deg; joints [-5.43, -0.746, 26.31, -63.672, 87.822, -51.763, -1798.36]
  MoveL 916 to (51.63, 282.88, 40) mm, rotated rx -180 ry -65 rz -166.1 deg; joints [-5.152, -0.204, 25.163, -63.539, 88.316, -52.194, -1803.9]
  MoveL 917 to (48.58, 287.83, 50) mm, rotated rx -180 ry -65 rz -160.19 deg; joints [-4.875, 0.396, 23.898, -63.412, 88.839, -52.677, -1809.813]
  MoveL 918 to (44.86, 292.68, 60) mm, rotated rx -180 ry -65 rz -153.93 deg; joints [-4.599, 1.074, 22.473, -63.291, 89.399, -53.23, -1816.069]
  MoveL 919 to (40.49, 297.28, 70) mm, rotated rx -180 ry -65 rz -147.36 deg; joints [-4.323, 1.865, 20.824, -63.179, 90.013, -53.883, -1822.636]
  MoveL 920 to (35.48, 301.51, 80) mm, rotated rx 180 ry -65 rz -140.52 deg; joints [-4.048, 2.832, 18.819, -63.081, 90.709, -54.694, -1829.477]
  MoveL 921 to (29.89, 305.25, 90) mm, rotated rx -180 ry -65 rz -133.45 deg; joints [-3.774, 4.15, 16.109, -63.005, 91.568, -55.819, -1836.554]
  MoveL 922 to (23.94, 308.16, 99.92) mm, rotated rx 180 ry -65 rz -126.18 deg; joints [-3.501, 7.137, 10.028, -63.027, 93.203, -58.46, -1843.825]
  MoveL 923 to (19.25, 308.72, 109.14) mm, rotated rx -180 ry -65 rz -118.76 deg; joints [-3.228, 7.118, 10.028, -62.941, 93.443, -58.36, -1851.243]
  MoveL 924 to (14.77, 308.97, 118.31) mm, rotated rx -180 ry -65 rz -111.24 deg; joints [-2.957, 7.1, 10.028, -62.855, 93.682, -58.257, -1858.761]
  MoveL 925 to (3.42, 313.28, 130) mm, rotated rx -180 ry -65 rz -113.67 deg; joints [-2.441, -1.054, 26.913, -59.966, 93.538, -59.269, -1866.327]
  MoveL 926 to (-3.62, 313.27, 140) mm, rotated rx -180 ry -65 rz -106.11 deg; joints [-2.168, -0.344, 25.451, -59.884, 94.128, -59.798, -1873.889]
  MoveL 927 to (-10.57, 312.43, 150) mm, rotated rx 180 ry -65 rz -98.61 deg; joints [-1.897, 0.468, 23.789, -59.818, 94.768, -60.411, -1881.395]
  MoveL 928 to (-17.28, 310.79, 160) mm, rotated rx 180 ry -65 rz -91.21 deg; joints [-1.626, 1.421, 21.845, -59.775, 95.481, -61.146, -1888.791]
  MoveL 929 to (-23.65, 308.43, 170) mm, rotated rx 180 ry -65 rz -83.97 deg; joints [-1.357, 2.601, 19.448, -59.767, 96.308, -62.077, -1896.03]
  MoveL 930 to (-29.57, 305.43, 180) mm, rotated rx -180 ry -65 rz -76.94 deg; joints [-1.089, 4.259, 16.089, -59.831, 97.38, -63.431, -1903.063]
  MoveL 931 to (-34, 302.1, 189.66) mm, rotated rx -180 ry -65 rz -70.15 deg; joints [-0.822, 7.255, 10.028, -60.112, 99.133, -65.984, -1909.847]
  MoveL 932 to (-35.74, 299.31, 198.51) mm, rotated rx -180 ry -65 rz -63.66 deg; joints [-0.556, 7.253, 10.028, -60.012, 99.354, -65.858, -1916.342]
  MoveL 933 to (-43.95, 293.72, 210) mm, rotated rx -180 ry -65 rz -67.49 deg; joints [-0.011, -1.288, 27.377, -56.827, 99.042, -66.776, -1922.509]
  MoveL 934 to (-47.51, 289.33, 220) mm, rotated rx -180 ry -65 rz -61.68 deg; joints [0.256, -0.443, 25.665, -56.81, 99.718, -67.377, -1928.316]
  MoveL 935 to (-50.46, 284.91, 230) mm, rotated rx -180 ry -65 rz -56.27 deg; joints [0.523, 0.519, 23.719, -56.821, 100.459, -68.08, -1933.731]
  MoveL 936 to (-52.84, 280.57, 240) mm, rotated rx -180 ry -65 rz -51.28 deg; joints [0.788, 1.654, 21.421, -56.876, 101.299, -68.937, -1938.724]
  MoveL 937 to (-54.69, 276.44, 250) mm, rotated rx 180 ry -65 rz -46.73 deg; joints [1.052, 3.098, 18.494, -57.008, 102.312, -70.069, -1943.267]
  MoveL 938 to (-56.08, 272.6, 260) mm, rotated rx -180 ry -65 rz -42.67 deg; joints [1.316, 5.488, 13.657, -57.363, 103.847, -72.043, -1947.333]
  MoveL 939 to (-55.45, 271.33, 268.93) mm, rotated rx -180 ry -65 rz -39.11 deg; joints [1.579, 7.278, 10.028, -57.645, 105.045, -73.506, -1950.894]
  MoveL 940 to (-57.77, 266.15, 280) mm, rotated rx -180 ry -65 rz -46.08 deg; joints [2.141, 15.899, -7.672, -59.572, 114.44, -90.293, -1953.924]
  MoveL 941 to (-58.22, 263.67, 290) mm, rotated rx 180 ry -65 rz -43.61 deg; joints [2.405, 14.999, -5.871, -59.121, 114.205, -89.297, -1956.394]
  MoveL 942 to (-78.63, 259.66, 290) mm, rotated rx -180 ry -65 rz -39.75 deg; joints [2.329, 13.048, -0.675, -57.958, 112.448, -86.325, -1960.245]
  Set speed (60.0 mm/s)
  MoveL 943 to (-78.34, 263.02, 280) mm, rotated rx -180 ry -65 rz -42.21 deg; joints [2.066, 14.303, -3.191, -58.516, 112.892, -87.633, -1957.792]
  MoveL 944 to (-77.78, 267.1, 270) mm, rotated rx -180 ry -65 rz -45.21 deg; joints [1.802, 15.351, -5.291, -59.005, 113.216, -88.757, -1954.787]
  MoveL 945 to (-76.86, 271.82, 260) mm, rotated rx 180 ry -65 rz -48.74 deg; joints [1.537, 16.266, -7.127, -59.448, 113.463, -89.765, -1951.259]
  MoveL 946 to (-72.8, 280.15, 248.46) mm, rotated rx -180 ry -65 rz -42.76 deg; joints [0.982, 7.902, 10.028, -57.768, 104.231, -73.275, -1947.238]
  MoveL 947 to (-73.09, 283.24, 239.78) mm, rotated rx 180 ry -65 rz -47.25 deg; joints [0.718, 7.906, 10.028, -57.882, 104.016, -73.409, -1942.753]
  MoveL 948 to (-70.88, 288.88, 230) mm, rotated rx -180 ry -65 rz -52.17 deg; joints [0.453, 11.32, 3.137, -58.774, 105.626, -76.609, -1937.833]
  MoveL 949 to (-67.49, 295.12, 220) mm, rotated rx 180 ry -65 rz -57.49 deg; joints [0.188, 12.968, -0.19, -59.286, 106.268, -78.243, -1932.509]
  MoveL 950 to (-63.28, 301.4, 210) mm, rotated rx -180 ry -65 rz -63.19 deg; joints [-0.079, 14.188, -2.65, -59.697, 106.674, -79.496, -1926.81]
  MoveL 951 to (-58.22, 307.54, 200) mm, rotated rx 180 ry -65 rz -69.23 deg; joints [-0.346, 15.195, -4.682, -60.056, 106.961, -80.559, -1920.77]
  MoveL 952 to (-52.31, 313.38, 190) mm, rotated rx -180 ry -65 rz -75.58 deg; joints [-0.614, 16.069, -6.441, -60.379, 107.172, -81.501, -1914.421]
  MoveL 953 to (-45.56, 318.73, 180) mm, rotated rx 180 ry -65 rz -82.2 deg; joints [-0.884, 16.846, -8.006, -60.676, 107.327, -82.356, -1907.8]
  MoveL 954 to (-34.96, 323.59, 168.97) mm, rotated rx -180 ry -65 rz -79.05 deg; joints [-1.419, 7.871, 10.028, -60.254, 98.333, -65.731, -1900.945]
  MoveL 955 to (-29.85, 327.37, 160) mm, rotated rx -180 ry -65 rz -86.1 deg; joints [-1.688, 7.661, 10.465, -60.327, 97.999, -65.66, -1893.897]
  MoveL 956 to (-21.11, 330.36, 150) mm, rotated rx -180 ry -65 rz -93.3 deg; joints [-1.957, 4.384, 17.101, -60.073, 96.108, -62.849, -1886.697]
  MoveL 957 to (-11.96, 332.32, 140) mm, rotated rx 180 ry -65 rz -100.61 deg; joints [-2.228, 2.979, 19.961, -60.063, 95.166, -61.708, -1879.391]
  MoveL 958 to (-2.59, 333.2, 130) mm, rotated rx -180 ry -65 rz -107.97 deg; joints [-2.499, 1.926, 22.113, -60.102, 94.401, -60.876, -1872.026]
  MoveL 959 to (6.83, 332.94, 120) mm, rotated rx 180 ry -65 rz -115.35 deg; joints [-2.772, 1.062, 23.89, -60.168, 93.732, -60.207, -1864.647]
  MoveL 960 to (16.13, 331.57, 110) mm, rotated rx -180 ry -65 rz -122.7 deg; joints [-3.046, 0.321, 25.422, -60.251, 93.124, -59.642, -1857.302]
  MoveL 961 to (25.11, 329.13, 100) mm, rotated rx 180 ry -65 rz -129.96 deg; joints [-3.32, -0.33, 26.777, -60.348, 92.561, -59.152, -1850.039]
  MoveL 962 to (37.13, 320.66, 88.23) mm, rotated rx -180 ry -65 rz -127.1 deg; joints [-3.827, 7.751, 10.028, -63.104, 92.647, -58.054, -1842.902]
  MoveL 963 to (43.23, 318.17, 78.97) mm, rotated rx -180 ry -65 rz -134.06 deg; joints [-4.1, 7.774, 10.028, -63.192, 92.405, -58.151, -1835.936]
  MoveL 964 to (49.15, 315.23, 69.66) mm, rotated rx 180 ry -65 rz -140.82 deg; joints [-4.374, 7.797, 10.028, -63.28, 92.161, -58.247, -1829.182]
  MoveL 965 to (55.08, 310.79, 60) mm, rotated rx -180 ry -65 rz -147.32 deg; joints [-4.649, 9.939, 5.751, -63.448, 92.884, -60.276, -1822.679]
  MoveL 966 to (60.61, 304.79, 50) mm, rotated rx -180 ry -65 rz -153.53 deg; joints [-4.924, 11.542, 2.562, -63.603, 93.352, -61.816, -1816.465]
  MoveL 967 to (65.29, 298.57, 40) mm, rotated rx 180 ry -65 rz -159.43 deg; joints [-5.201, 12.63, 0.417, -63.733, 93.58, -62.885, -1810.575]
  MoveL 968 to (69.12, 292.29, 30) mm, rotated rx -180 ry -65 rz -164.96 deg; joints [-5.478, 13.504, -1.298, -63.849, 93.709, -63.76, -1805.041]
  MoveL 969 to (72.16, 286.11, 20) mm, rotated rx 180 ry -65 rz -170.1 deg; joints [-5.755, 14.253, -2.76, -63.955, 93.779, -64.522, -1799.895]
  MoveL 970 to (74.48, 280.19, 10) mm, rotated rx 180 ry -65 rz -174.83 deg; joints [-6.033, 14.916, -4.051, -64.055, 93.809, -65.208, -1795.168]
  MoveL 971 to (76.17, 274.65, 0) mm, rotated rx -180 ry -65 rz -179.11 deg; joints [-6.312, 15.517, -5.217, -64.148, 93.809, -65.837, -1790.889]
  MoveL 972 to (-78.63, 259.66, 290) mm, rotated rx -180 ry -65 rz -39.75 deg; joints [2.329, 13.048, -0.675, -57.958, 112.448, -86.325, -1960.245]
  Set speed (60.0 mm/s)
  MoveL 973 to (-58.93, 252.99, 290) mm, rotated rx -180 ry -65 rz -33.22 deg; joints [2.401, 14.923, -5.655, -59.069, 114.13, -89.167, -1966.784]
  MoveL 974 to (76.17, 274.65, 0) mm, rotated rx 180 ry -65 rz -179.11 deg; joints [-6.312, 15.517, -5.217, -64.148, 93.809, -65.837, -1790.889]
  Set speed (60.0 mm/s)
  MoveL 975 to (54.99, 272.92, -0.43) mm, rotated rx -180 ry -65 rz -165.16 deg; joints [-6.453, 6.969, 10.028, -66.346, 87.28, -50.763, -1794.838]
  MoveL 976 to (76.17, 274.65, 0) mm, rotated rx 180 ry -65 rz -179.11 deg; joints [-6.312, 0.429, 25.273, -64.043, 87.048, -51.99, -1790.889]
  Set speed (60.0 mm/s)
  MoveL 977 to (74.48, 280.19, 10) mm, rotated rx -180 ry -65 rz -174.83 deg; joints [-6.033, 0.983, 24.107, -63.903, 87.543, -52.431, -1795.168]
  MoveL 978 to (72.16, 286.11, 20) mm, rotated rx 180 ry -65 rz -170.1 deg; joints [-5.755, 1.597, 22.816, -63.768, 88.068, -52.927, -1799.895]
  MoveL 979 to (69.12, 292.29, 30) mm, rotated rx -180 ry -65 rz -164.96 deg; joints [-5.478, 2.295, 21.353, -63.638, 88.634, -53.5, -1805.041]
  MoveL 980 to (65.29, 298.57, 40) mm, rotated rx -180 ry -65 rz -159.43 deg; joints [-5.201, 3.118, 19.638, -63.516, 89.259, -54.186, -1810.575]
  MoveL 981 to (60.61, 304.79, 50) mm, rotated rx -180 ry -65 rz -153.53 deg; joints [-4.924, 4.154, 17.493, -63.406, 89.983, -55.064, -1816.465]
  MoveL 982 to (55.08, 310.79, 60) mm, rotated rx 180 ry -65 rz -147.32 deg; joints [-4.649, 5.706, 14.305, -63.319, 90.947, -56.411, -1822.679]
  MoveL 983 to (49.15, 315.23, 69.66) mm, rotated rx -180 ry -65 rz -140.82 deg; joints [-4.374, 7.797, 10.028, -63.28, 92.161, -58.247, -1829.182]
  MoveL 984 to (43.23, 318.17, 78.97) mm, rotated rx -180 ry -65 rz -134.06 deg; joints [-4.1, 7.774, 10.028, -63.192, 92.405, -58.151, -1835.936]
  MoveL 985 to (37.13, 320.66, 88.23) mm, rotated rx 180 ry -65 rz -127.1 deg; joints [-3.827, 7.751, 10.028, -63.104, 92.647, -58.054, -1842.902]
  MoveL 986 to (25.11, 329.13, 100) mm, rotated rx -180 ry -65 rz -129.96 deg; joints [-3.32, 16.246, -6.721, -62.092, 100.755, -74.073, -1850.039]
  MoveL 987 to (16.13, 331.57, 110) mm, rotated rx -180 ry -65 rz -122.7 deg; joints [-3.046, 15.556, -5.366, -61.909, 100.682, -73.346, -1857.302]
  MoveL 988 to (6.83, 332.94, 120) mm, rotated rx -180 ry -65 rz -115.35 deg; joints [-2.772, 14.781, -3.834, -61.71, 100.561, -72.538, -1864.647]
  MoveL 989 to (-2.59, 333.2, 130) mm, rotated rx -180 ry -65 rz -107.97 deg; joints [-2.499, 13.887, -2.057, -61.489, 100.377, -71.618, -1872.026]
  MoveL 990 to (-11.96, 332.32, 140) mm, rotated rx 180 ry -65 rz -100.61 deg; joints [-2.228, 12.81, 0.095, -61.238, 100.094, -70.531, -1879.391]
  MoveL 991 to (-21.11, 330.36, 150) mm, rotated rx 180 ry -65 rz -93.3 deg; joints [-1.957, 11.385, 2.954, -60.934, 99.631, -69.127, -1886.697]
  MoveL 992 to (-29.85, 327.37, 160) mm, rotated rx -180 ry -65 rz -86.1 deg; joints [-1.688, 8.093, 9.591, -60.382, 98.217, -66.047, -1893.897]
  MoveL 993 to (-34.96, 323.59, 168.97) mm, rotated rx -180 ry -65 rz -79.05 deg; joints [-1.419, 7.871, 10.028, -60.254, 98.333, -65.731, -1900.945]
  MoveL 994 to (-45.56, 318.73, 180) mm, rotated rx 180 ry -65 rz -82.2 deg; joints [-0.884, -1.001, 28.062, -57.16, 97.858, -66.382, -1907.8]
  MoveL 995 to (-52.31, 313.38, 190) mm, rotated rx -180 ry -65 rz -75.58 deg; joints [-0.614, -0.23, 26.497, -57.116, 98.491, -66.924, -1914.421]
  MoveL 996 to (-58.22, 307.54, 200) mm, rotated rx -180 ry -65 rz -69.23 deg; joints [-0.346, 0.638, 24.738, -57.095, 99.178, -67.549, -1920.77]
  MoveL 997 to (-63.28, 301.4, 210) mm, rotated rx -180 ry -65 rz -63.19 deg; joints [-0.079, 1.641, 22.706, -57.106, 99.94, -68.291, -1926.81]
  MoveL 998 to (-67.49, 295.12, 220) mm, rotated rx -180 ry -65 rz -57.49 deg; joints [0.188, 2.856, 20.246, -57.166, 100.821, -69.219, -1932.509]
  MoveL 999 to (-70.88, 288.88, 230) mm, rotated rx 180 ry -65 rz -52.17 deg; joints [0.453, 4.5, 16.919, -57.324, 101.938, -70.528, -1937.833]
  MoveL 1000 to (-73.09, 283.24, 239.78) mm, rotated rx 180 ry -65 rz -47.25 deg; joints [0.718, 7.906, 10.028, -57.882, 104.016, -73.409, -1942.753]
  MoveL 1001 to (-72.8, 280.15, 248.46) mm, rotated rx -180 ry -65 rz -42.76 deg; joints [0.982, 7.902, 10.028, -57.768, 104.231, -73.275, -1947.238]
  MoveL 1002 to (-76.86, 271.82, 260) mm, rotated rx -180 ry -65 rz -48.74 deg; joints [1.537, -0.712, 27.183, -54.488, 103.955, -74.436, -1951.259]
  MoveL 1003 to (-77.78, 267.1, 270) mm, rotated rx 180 ry -65 rz -45.21 deg; joints [1.802, 0.19, 25.347, -54.531, 104.691, -75.079, -1954.787]
  MoveL 1004 to (-78.34, 263.02, 280) mm, rotated rx -180 ry -65 rz -42.21 deg; joints [2.066, 1.221, 23.247, -54.617, 105.506, -75.837, -1957.792]
  MoveL 1005 to (-78.63, 259.66, 290) mm, rotated rx 180 ry -65 rz -39.75 deg; joints [2.329, 2.455, 20.731, -54.77, 106.443, -76.78, -1960.245]
  MoveL 1006 to (-58.93, 252.99, 290) mm, rotated rx -180 ry -65 rz -33.22 deg; joints [2.401, -0.598, 25.711, -54.282, 105.378, -75.109, -1966.784]
  Set speed (60.0 mm/s)
  MoveL 1007 to (-58.94, 255.51, 280) mm, rotated rx -180 ry -65 rz -35.64 deg; joints [2.137, -1.491, 27.534, -54.231, 104.642, -74.471, -1964.356]
  MoveL 1008 to (-57.41, 261.39, 268.77) mm, rotated rx 180 ry -65 rz -28.62 deg; joints [1.575, 7.309, 10.028, -57.64, 105.026, -73.481, -1961.378]
  MoveL 1009 to (-58.44, 262.16, 260) mm, rotated rx -180 ry -65 rz -32.12 deg; joints [1.313, 8.562, 7.507, -58.045, 105.488, -74.733, -1957.879]
  MoveL 1010 to (-57.77, 266.19, 250) mm, rotated rx 180 ry -65 rz -36.12 deg; joints [1.049, 11.306, 1.97, -58.838, 106.732, -77.349, -1953.884]
  MoveL 1011 to (-56.69, 270.59, 240) mm, rotated rx 180 ry -65 rz -40.58 deg; joints [0.785, 12.813, -1.07, -59.338, 107.298, -78.863, -1949.42]
  MoveL 1012 to (-55.14, 275.28, 230) mm, rotated rx 180 ry -65 rz -45.49 deg; joints [0.519, 13.979, -3.425, -59.754, 107.676, -80.075, -1944.512]
  MoveL 1013 to (-53.04, 280.16, 220) mm, rotated rx 180 ry -65 rz -50.81 deg; joints [0.253, 14.962, -5.409, -60.121, 107.952, -81.124, -1939.189]
  MoveL 1014 to (-50.33, 285.12, 210) mm, rotated rx -180 ry -65 rz -56.52 deg; joints [-0.014, 15.824, -7.151, -60.455, 108.158, -82.065, -1933.477]
  MoveL 1015 to (-43.01, 292.31, 198.4) mm, rotated rx 180 ry -65 rz -52.6 deg; joints [-0.558, 7.277, 10.028, -60.01, 99.34, -65.838, -1927.405]
  MoveL 1016 to (-41.79, 295.3, 189.56) mm, rotated rx -180 ry -65 rz -59 deg; joints [-0.824, 7.277, 10.028, -60.11, 99.12, -65.966, -1921.005]
  MoveL 1017 to (-38.31, 299.24, 180) mm, rotated rx -180 ry -65 rz -65.69 deg; joints [-1.091, 4.461, 15.72, -59.851, 97.463, -63.578, -1914.31]
  MoveL 1018 to (-33.03, 303.26, 170) mm, rotated rx -180 ry -65 rz -72.64 deg; joints [-1.359, 2.714, 19.252, -59.776, 96.349, -62.15, -1907.357]
  MoveL 1019 to (-27.19, 306.74, 160) mm, rotated rx -180 ry -65 rz -79.81 deg; joints [-1.628, 1.495, 21.722, -59.78, 95.504, -61.189, -1900.187]
  MoveL 1020 to (-20.88, 309.56, 150) mm, rotated rx -180 ry -65 rz -87.16 deg; joints [-1.898, 0.514, 23.714, -59.821, 94.782, -60.436, -1892.844]
  MoveL 1021 to (-14.2, 311.65, 140) mm, rotated rx 180 ry -65 rz -94.63 deg; joints [-2.169, -0.32, 25.413, -59.885, 94.135, -59.81, -1885.374]
  MoveL 1022 to (-7.28, 312.93, 130) mm, rotated rx 180 ry -65 rz -102.17 deg; joints [-2.441, -1.049, 26.905, -59.966, 93.54, -59.272, -1877.828]
  MoveL 1023 to (4.68, 310.86, 118.32) mm, rotated rx 180 ry -65 rz -99.74 deg; joints [-2.957, 7.097, 10.028, -62.855, 93.684, -58.259, -1870.258]
  MoveL 1024 to (9.07, 311.4, 109.17) mm, rotated rx -180 ry -65 rz -107.29 deg; joints [-3.228, 7.111, 10.028, -62.941, 93.447, -58.366, -1862.715]
  MoveL 1025 to (13.72, 311.7, 99.96) mm, rotated rx -180 ry -65 rz -114.75 deg; joints [-3.5, 7.127, 10.028, -63.028, 93.208, -58.47, -1855.252]
  MoveL 1026 to (20.21, 309.81, 90) mm, rotated rx -180 ry -65 rz -122.08 deg; joints [-3.773, 10.284, 3.685, -63.298, 94.412, -61.438, -1847.921]
  MoveL 1027 to (26.38, 307.15, 80) mm, rotated rx 180 ry -65 rz -129.23 deg; joints [-4.046, 11.627, 1.012, -63.466, 94.77, -62.75, -1840.769]
  MoveL 1028 to (32.08, 303.89, 70) mm, rotated rx -180 ry -65 rz -136.16 deg; joints [-4.321, 12.635, -0.983, -63.609, 94.969, -63.756, -1833.843]
  MoveL 1029 to (37.21, 300.16, 60) mm, rotated rx -180 ry -65 rz -142.82 deg; joints [-4.597, 13.472, -2.627, -63.737, 95.085, -64.603, -1827.185]
  MoveL 1030 to (41.73, 296.07, 50) mm, rotated rx 180 ry -65 rz -149.17 deg; joints [-4.873, 14.199, -4.048, -63.854, 95.147, -65.349, -1820.833]
  MoveL 1031 to (45.64, 291.75, 40) mm, rotated rx 180 ry -65 rz -155.18 deg; joints [-5.15, 14.848, -5.31, -63.962, 95.172, -66.022, -1814.824]
  MoveL 1032 to (48.92, 287.33, 30) mm, rotated rx -180 ry -65 rz -160.81 deg; joints [-5.428, 15.438, -6.453, -64.063, 95.168, -66.642, -1809.19]
  MoveL 1033 to (51.27, 276.9, 18.49) mm, rotated rx 180 ry -65 rz -156.04 deg; joints [-5.901, 6.925, 10.028, -66.192, 87.781, -50.591, -1803.962]
  MoveL 1034 to (53.19, 274.81, 9.05) mm, rotated rx -180 ry -65 rz -160.83 deg; joints [-6.177, 6.948, 10.028, -66.269, 87.531, -50.676, -1799.169]
  MoveL 1035 to (54.99, 272.92, -0.43) mm, rotated rx 180 ry -65 rz -165.16 deg; joints [-6.453, 6.969, 10.028, -66.346, 87.28, -50.763, -1794.838]
  MoveL 1036 to (-58.93, 252.99, 290) mm, rotated rx 180 ry -65 rz -33.22 deg; joints [2.401, 14.923, -5.655, -59.069, 114.13, -89.167, -1966.784]
  Set speed (60.0 mm/s)
  MoveL 1037 to (-37.11, 208.63, 290) mm, rotated rx -180 ry -65 rz 14.16 deg; joints [2.386, 14.605, -4.762, -58.856, 113.821, -88.637, -2014.156]
  MoveL 1038 to (55.37, 274.67, 0) mm, rotated rx 180 ry -65 rz -175.16 deg; joints [-6.265, 16.96, -9.386, -64.329, 95.037, -68.28, -2154.838]
  Set speed (60.0 mm/s)
  MoveL 1039 to (20.67, 309.5, -0.07) mm, rotated rx -180 ry -65 rz -112.4 deg; joints [-6.445, 6.863, 10.028, -66.339, 87.33, -50.857, -2207.595]
  MoveL 1040 to (54.99, 272.92, -0.43) mm, rotated rx 180 ry -65 rz -165.16 deg; joints [-6.453, 6.969, 10.028, -66.346, 87.28, -50.763, -2154.838]
  Set speed (60.0 mm/s)
  MoveL 1041 to (53.19, 274.81, 9.05) mm, rotated rx -180 ry -65 rz -160.83 deg; joints [-6.177, 6.948, 10.028, -66.269, 87.531, -50.676, -2159.169]
  MoveL 1042 to (51.27, 276.9, 18.49) mm, rotated rx 180 ry -65 rz -156.04 deg; joints [-5.901, 6.925, 10.028, -66.192, 87.781, -50.591, -2163.962]
  MoveL 1043 to (48.92, 287.33, 30) mm, rotated rx -180 ry -65 rz -160.81 deg; joints [-5.428, 15.438, -6.453, -64.063, 95.168, -66.642, -2169.19]
  MoveL 1044 to (45.64, 291.75, 40) mm, rotated rx 180 ry -65 rz -155.18 deg; joints [-5.15, 14.848, -5.31, -63.962, 95.172, -66.022, -2174.824]
  MoveL 1045 to (41.73, 296.07, 50) mm, rotated rx -180 ry -65 rz -149.17 deg; joints [-4.873, 14.199, -4.048, -63.854, 95.147, -65.349, -2180.833]
  MoveL 1046 to (37.21, 300.16, 60) mm, rotated rx -180 ry -65 rz -142.82 deg; joints [-4.597, 13.472, -2.627, -63.737, 95.085, -64.603, -2187.185]
  MoveL 1047 to (32.08, 303.89, 70) mm, rotated rx 180 ry -65 rz -136.16 deg; joints [-4.321, 12.635, -0.983, -63.609, 94.969, -63.756, -2193.843]
  MoveL 1048 to (26.38, 307.15, 80) mm, rotated rx 180 ry -65 rz -129.23 deg; joints [-4.046, 11.627, 1.012, -63.466, 94.77, -62.75, -2200.769]
  MoveL 1049 to (20.21, 309.81, 90) mm, rotated rx 180 ry -65 rz -122.08 deg; joints [-3.773, 10.284, 3.685, -63.298, 94.412, -61.438, -2207.921]
  MoveL 1050 to (13.72, 311.7, 99.96) mm, rotated rx -180 ry -65 rz -114.75 deg; joints [-3.5, 7.127, 10.028, -63.028, 93.208, -58.47, -2215.252]
  MoveL 1051 to (9.07, 311.4, 109.17) mm, rotated rx -180 ry -65 rz -107.29 deg; joints [-3.228, 7.111, 10.028, -62.941, 93.447, -58.366, -2222.715]
  MoveL 1052 to (4.68, 310.86, 118.32) mm, rotated rx -180 ry -65 rz -99.74 deg; joints [-2.957, 7.097, 10.028, -62.855, 93.684, -58.259, -2230.258]
  MoveL 1053 to (-7.28, 312.93, 130) mm, rotated rx 180 ry -65 rz -102.17 deg; joints [-2.441, 15.654, -6.85, -61.997, 101.86, -74.306, -2237.828]
  MoveL 1054 to (-14.2, 311.65, 140) mm, rotated rx -180 ry -65 rz -94.63 deg; joints [-2.169, 14.907, -5.357, -61.79, 101.746, -73.506, -2245.374]
  MoveL 1055 to (-20.88, 309.56, 150) mm, rotated rx -180 ry -65 rz -87.16 deg; joints [-1.898, 14.059, -3.659, -61.562, 101.577, -72.611, -2252.844]
  MoveL 1056 to (-27.19, 306.74, 160) mm, rotated rx 180 ry -65 rz -79.81 deg; joints [-1.628, 13.069, -1.666, -61.307, 101.331, -71.584, -2260.187]
  MoveL 1057 to (-33.03, 303.26, 170) mm, rotated rx -180 ry -65 rz -72.64 deg; joints [-1.359, 11.844, 0.804, -61.012, 100.96, -70.343, -2267.357]
  MoveL 1058 to (-38.31, 299.24, 180) mm, rotated rx -180 ry -65 rz -65.69 deg; joints [-1.091, 10.094, 4.336, -60.633, 100.319, -68.63, -2274.31]
  MoveL 1059 to (-41.79, 295.3, 189.56) mm, rotated rx -180 ry -65 rz -59 deg; joints [-0.824, 7.277, 10.028, -60.11, 99.12, -65.966, -2281.005]
  MoveL 1060 to (-43.01, 292.31, 198.4) mm, rotated rx 180 ry -65 rz -52.6 deg; joints [-0.558, 7.277, 10.028, -60.01, 99.34, -65.838, -2287.405]
  MoveL 1061 to (-50.33, 285.12, 210) mm, rotated rx -180 ry -65 rz -56.52 deg; joints [-0.014, -1.177, 27.206, -56.837, 99.072, -66.828, -2293.477]
  MoveL 1062 to (-53.04, 280.16, 220) mm, rotated rx -180 ry -65 rz -50.81 deg; joints [0.253, -0.316, 25.465, -56.822, 99.755, -67.441, -2299.189]
  MoveL 1063 to (-55.14, 275.28, 230) mm, rotated rx 180 ry -65 rz -45.49 deg; joints [0.519, 0.665, 23.481, -56.837, 100.507, -68.16, -2304.512]
  MoveL 1064 to (-56.69, 270.59, 240) mm, rotated rx 180 ry -65 rz -40.58 deg; joints [0.785, 1.829, 21.126, -56.898, 101.362, -69.04, -2309.42]
  MoveL 1065 to (-57.77, 266.19, 250) mm, rotated rx 180 ry -65 rz -36.12 deg; joints [1.049, 3.331, 18.086, -57.042, 102.405, -70.222, -2313.884]
  MoveL 1066 to (-58.44, 262.16, 260) mm, rotated rx -180 ry -65 rz -32.12 deg; joints [1.313, 6.067, 12.549, -57.475, 104.129, -72.505, -2317.879]
  MoveL 1067 to (-57.41, 261.39, 268.77) mm, rotated rx 180 ry -65 rz -28.62 deg; joints [1.575, 7.309, 10.028, -57.64, 105.026, -73.481, -2321.378]
  MoveL 1068 to (-58.94, 255.51, 280) mm, rotated rx 180 ry -65 rz -35.64 deg; joints [2.137, 15.834, -7.478, -59.523, 114.371, -90.173, -2324.356]
  MoveL 1069 to (-58.93, 252.99, 290) mm, rotated rx 180 ry -65 rz -33.22 deg; joints [2.401, 14.923, -5.655, -59.069, 114.13, -89.167, -2326.784]
  MoveL 1070 to (-37.11, 208.63, 290) mm, rotated rx 180 ry -65 rz 14.16 deg; joints [2.386, 14.605, -4.762, -58.856, 113.821, -88.637, -2374.156]
  Set speed (60.0 mm/s)
  MoveL 1071 to (-39.03, 210.26, 280) mm, rotated rx 180 ry -65 rz 11.88 deg; joints [2.122, 15.557, -6.662, -59.32, 114.084, -89.673, -2371.877]
  MoveL 1072 to (-43.03, 216.88, 268.1) mm, rotated rx 180 ry -65 rz 19.09 deg; joints [1.56, 7.436, 10.028, -57.618, 104.945, -73.378, -2369.089]
  MoveL 1073 to (-44.2, 216.27, 259.47) mm, rotated rx 180 ry -65 rz 15.82 deg; joints [1.297, 7.446, 10.028, -57.73, 104.728, -73.508, -2365.82]
  MoveL 1074 to (-46.4, 218.08, 250) mm, rotated rx 180 ry -65 rz 12.1 deg; joints [1.034, 10.364, 4.146, -58.533, 106.078, -76.258, -2362.097]
  MoveL 1075 to (-49.06, 221.75, 240) mm, rotated rx -180 ry -65 rz 7.95 deg; joints [0.769, 12.208, 0.431, -59.108, 106.827, -78.066, -2357.947]
  MoveL 1076 to (-51.62, 225.97, 230) mm, rotated rx -180 ry -65 rz 3.4 deg; joints [0.504, 13.51, -2.192, -59.552, 107.277, -79.393, -2353.396]
  MoveL 1077 to (-53.98, 230.73, 220) mm, rotated rx -180 ry -65 rz -1.53 deg; joints [0.237, 14.573, -4.335, -59.936, 107.596, -80.509, -2348.469]
  MoveL 1078 to (-56, 236.01, 210) mm, rotated rx 180 ry -65 rz -6.81 deg; joints [-0.029, 15.49, -6.188, -60.282, 107.834, -81.498, -2343.192]
  MoveL 1079 to (-57.57, 241.75, 200) mm, rotated rx 180 ry -65 rz -12.41 deg; joints [-0.297, 16.307, -7.841, -60.601, 108.016, -82.4, -2337.589]
  MoveL 1080 to (-57.7, 250.93, 188.91) mm, rotated rx 180 ry -65 rz -8.32 deg; joints [-0.838, 7.415, 10.028, -60.096, 99.04, -65.853, -2331.684]
  MoveL 1081 to (-58.95, 254.32, 180) mm, rotated rx -180 ry -65 rz -14.5 deg; joints [-1.105, 6.676, 11.512, -60.098, 98.448, -65.326, -2325.504]
  MoveL 1082 to (-58.59, 260.95, 170) mm, rotated rx -180 ry -65 rz -20.93 deg; joints [-1.372, 3.692, 17.533, -59.854, 96.711, -62.801, -2319.073]
  MoveL 1083 to (-57.45, 267.65, 160) mm, rotated rx -180 ry -65 rz -27.58 deg; joints [-1.64, 2.212, 20.512, -59.827, 95.743, -61.623, -2312.419]
  MoveL 1084 to (-55.51, 274.28, 150) mm, rotated rx -180 ry -65 rz -34.43 deg; joints [-1.908, 1.08, 22.789, -59.852, 94.954, -60.753, -2305.573]
  MoveL 1085 to (-52.77, 280.72, 140) mm, rotated rx 180 ry -65 rz -41.43 deg; joints [-2.178, 0.132, 24.692, -59.907, 94.262, -60.047, -2298.565]
  MoveL 1086 to (-49.26, 286.82, 130) mm, rotated rx -180 ry -65 rz -48.57 deg; joints [-2.449, -0.693, 26.35, -59.981, 93.633, -59.448, -2291.431]
  MoveL 1087 to (-45.04, 292.47, 120) mm, rotated rx 180 ry -65 rz -55.79 deg; joints [-2.72, -1.428, 27.828, -60.07, 93.051, -58.926, -2284.209]
  MoveL 1088 to (-36.93, 298.71, 108.97) mm, rotated rx -180 ry -65 rz -53.06 deg; joints [-3.232, 7.159, 10.028, -62.94, 93.422, -58.325, -2276.94]
  MoveL 1089 to (-34.29, 302.11, 99.84) mm, rotated rx -180 ry -65 rz -60.33 deg; joints [-3.502, 7.157, 10.028, -63.027, 93.192, -58.443, -2269.668]
  MoveL 1090 to (-29.06, 305.72, 90) mm, rotated rx 180 ry -65 rz -67.56 deg; joints [-3.774, 10.181, 3.919, -63.289, 94.352, -61.321, -2262.441]
  MoveL 1091 to (-23.03, 308.7, 80) mm, rotated rx 180 ry -65 rz -74.69 deg; joints [-4.046, 11.652, 0.95, -63.469, 94.786, -62.782, -2255.308]
  MoveL 1092 to (-16.86, 310.92, 70) mm, rotated rx -180 ry -65 rz -81.68 deg; joints [-4.319, 12.725, -1.209, -63.62, 95.031, -63.878, -2248.32]
  MoveL 1093 to (-10.69, 312.41, 60) mm, rotated rx 180 ry -65 rz -88.47 deg; joints [-4.593, 13.603, -2.969, -63.754, 95.181, -64.792, -2241.529]
  MoveL 1094 to (-4.64, 313.2, 50) mm, rotated rx -180 ry -65 rz -95.02 deg; joints [-4.869, 14.357, -4.476, -63.875, 95.27, -65.59, -2234.983]
  MoveL 1095 to (1.18, 313.37, 40) mm, rotated rx -180 ry -65 rz -101.27 deg; joints [-5.145, 15.025, -5.805, -63.987, 95.316, -66.306, -2228.733]
  MoveL 1096 to (6.67, 313.01, 30) mm, rotated rx -180 ry -65 rz -107.17 deg; joints [-5.421, 15.628, -6.998, -64.091, 95.329, -66.96, -2222.826]
  MoveL 1097 to (15.43, 309.15, 18.81) mm, rotated rx 180 ry -65 rz -102.69 deg; joints [-5.894, 6.836, 10.028, -66.187, 87.823, -50.67, -2217.306]
  MoveL 1098 to (18.15, 309.3, 9.39) mm, rotated rx -180 ry -65 rz -107.78 deg; joints [-6.169, 6.849, 10.028, -66.263, 87.577, -50.764, -2212.216]
  MoveL 1099 to (20.67, 309.5, -0.07) mm, rotated rx -180 ry -65 rz -112.4 deg; joints [-6.445, 6.863, 10.028, -66.339, 87.33, -50.857, -2207.595]
  MoveL 1100 to (-37.11, 208.63, 290) mm, rotated rx 180 ry -65 rz 14.16 deg; joints [2.386, 14.605, -4.762, -58.856, 113.821, -88.637, -2374.156]
  Set speed (60.0 mm/s)
  MoveL 1101 to (-43.85, 188.95, 290) mm, rotated rx -180 ry -65 rz 18.32 deg; joints [2.311, 12.354, 1.025, -57.619, 111.896, -85.415, -2378.321]
  MoveL 1102 to (20.67, 309.5, -0.07) mm, rotated rx 180 ry -65 rz -112.4 deg; joints [-6.445, 6.863, 10.028, -66.339, 87.33, -50.857, -2207.595]
  Set speed (60.0 mm/s)
  MoveL 1103 to (20.57, 330.51, 0) mm, rotated rx 180 ry -65 rz -116.27 deg; joints [-6.302, -0.161, 26.213, -64.056, 86.902, -51.671, -2213.733]
  MoveL 1104 to (20.67, 309.5, -0.07) mm, rotated rx -180 ry -65 rz -112.4 deg; joints [-6.445, 6.863, 10.028, -66.339, 87.33, -50.857, -2207.595]
  Set speed (60.0 mm/s)
  MoveL 1105 to (18.15, 309.3, 9.39) mm, rotated rx 180 ry -65 rz -107.78 deg; joints [-6.169, 6.849, 10.028, -66.263, 87.577, -50.764, -2212.216]
  MoveL 1106 to (15.43, 309.15, 18.81) mm, rotated rx 180 ry -65 rz -102.69 deg; joints [-5.894, 6.836, 10.028, -66.187, 87.823, -50.67, -2217.306]
  MoveL 1107 to (6.67, 313.01, 30) mm, rotated rx -180 ry -65 rz -107.17 deg; joints [-5.421, 15.628, -6.998, -64.091, 95.329, -66.96, -2222.826]
  MoveL 1108 to (1.18, 313.37, 40) mm, rotated rx -180 ry -65 rz -101.27 deg; joints [-5.145, 15.025, -5.805, -63.987, 95.316, -66.306, -2228.733]
  MoveL 1109 to (-4.64, 313.2, 50) mm, rotated rx 180 ry -65 rz -95.02 deg; joints [-4.869, 14.357, -4.476, -63.875, 95.27, -65.59, -2234.983]
  MoveL 1110 to (-10.69, 312.41, 60) mm, rotated rx -180 ry -65 rz -88.47 deg; joints [-4.593, 13.603, -2.969, -63.754, 95.181, -64.792, -2241.529]
  MoveL 1111 to (-16.86, 310.92, 70) mm, rotated rx -180 ry -65 rz -81.68 deg; joints [-4.319, 12.725, -1.209, -63.62, 95.031, -63.878, -2248.32]
  MoveL 1112 to (-23.03, 308.7, 80) mm, rotated rx -180 ry -65 rz -74.69 deg; joints [-4.046, 11.652, 0.95, -63.469, 94.786, -62.782, -2255.308]
  MoveL 1113 to (-29.06, 305.72, 90) mm, rotated rx 180 ry -65 rz -67.56 deg; joints [-3.774, 10.181, 3.919, -63.289, 94.352, -61.321, -2262.441]
  MoveL 1114 to (-34.29, 302.11, 99.84) mm, rotated rx 180 ry -65 rz -60.33 deg; joints [-3.502, 7.157, 10.028, -63.027, 93.192, -58.443, -2269.668]
  MoveL 1115 to (-36.93, 298.71, 108.97) mm, rotated rx 180 ry -65 rz -53.06 deg; joints [-3.232, 7.159, 10.028, -62.94, 93.422, -58.325, -2276.94]
  MoveL 1116 to (-45.04, 292.47, 120) mm, rotated rx -180 ry -65 rz -55.79 deg; joints [-2.72, -1.428, 27.828, -60.07, 93.051, -58.926, -2284.209]
  MoveL 1117 to (-49.26, 286.82, 130) mm, rotated rx -180 ry -65 rz -48.57 deg; joints [-2.449, -0.693, 26.35, -59.981, 93.633, -59.448, -2291.431]
  MoveL 1118 to (-52.77, 280.72, 140) mm, rotated rx 180 ry -65 rz -41.43 deg; joints [-2.178, 0.132, 24.692, -59.907, 94.262, -60.047, -2298.565]
  MoveL 1119 to (-55.51, 274.28, 150) mm, rotated rx -180 ry -65 rz -34.43 deg; joints [-1.908, 1.08, 22.789, -59.852, 94.954, -60.753, -2305.573]
  MoveL 1120 to (-57.45, 267.65, 160) mm, rotated rx -180 ry -65 rz -27.58 deg; joints [-1.64, 2.212, 20.512, -59.827, 95.743, -61.623, -2312.419]
  MoveL 1121 to (-58.59, 260.95, 170) mm, rotated rx -180 ry -65 rz -20.93 deg; joints [-1.372, 3.692, 17.533, -59.854, 96.711, -62.801, -2319.073]
  MoveL 1122 to (-58.95, 254.32, 180) mm, rotated rx -180 ry -65 rz -14.5 deg; joints [-1.105, 6.676, 11.512, -60.098, 98.448, -65.326, -2325.504]
  MoveL 1123 to (-57.7, 250.93, 188.91) mm, rotated rx -180 ry -65 rz -8.32 deg; joints [-0.838, 7.415, 10.028, -60.096, 99.04, -65.853, -2331.684]
  MoveL 1124 to (-57.57, 241.75, 200) mm, rotated rx -180 ry -65 rz -12.41 deg; joints [-0.297, -1.377, 27.897, -56.92, 98.591, -66.552, -2337.589]
  MoveL 1125 to (-56, 236.01, 210) mm, rotated rx 180 ry -65 rz -6.81 deg; joints [-0.029, -0.558, 26.244, -56.891, 99.248, -67.127, -2343.192]
  MoveL 1126 to (-53.98, 230.73, 220) mm, rotated rx -180 ry -65 rz -1.53 deg; joints [0.237, 0.358, 24.391, -56.888, 99.962, -67.789, -2348.469]
  MoveL 1127 to (-51.62, 225.97, 230) mm, rotated rx -180 ry -65 rz 3.4 deg; joints [0.504, 1.416, 22.248, -56.921, 100.758, -68.578, -2353.396]
  MoveL 1128 to (-49.06, 221.75, 240) mm, rotated rx 180 ry -65 rz 7.95 deg; joints [0.769, 2.71, 19.625, -57.012, 101.688, -69.579, -2357.947]
  MoveL 1129 to (-46.4, 218.08, 250) mm, rotated rx 180 ry -65 rz 12.1 deg; joints [1.034, 4.542, 15.91, -57.231, 102.916, -71.06, -2362.097]
  MoveL 1130 to (-44.2, 216.27, 259.47) mm, rotated rx -180 ry -65 rz 15.82 deg; joints [1.297, 7.446, 10.028, -57.73, 104.728, -73.508, -2365.82]
  MoveL 1131 to (-43.03, 216.88, 268.1) mm, rotated rx 180 ry -65 rz 19.09 deg; joints [1.56, 7.436, 10.028, -57.618, 104.945, -73.378, -2369.089]
  MoveL 1132 to (-39.03, 210.26, 280) mm, rotated rx 180 ry -65 rz 11.88 deg; joints [2.122, -0.96, 26.718, -54.301, 104.797, -74.72, -2371.877]
  MoveL 1133 to (-37.11, 208.63, 290) mm, rotated rx -180 ry -65 rz 14.16 deg; joints [2.386, -0.033, 24.818, -54.365, 105.558, -75.393, -2374.156]
  MoveL 1134 to (-43.85, 188.95, 290) mm, rotated rx -180 ry -65 rz 18.32 deg; joints [2.311, 3.444, 19.031, -54.954, 106.839, -77.397, -2378.321]
  Set speed (60.0 mm/s)
  MoveL 1135 to (-46.6, 190.89, 280) mm, rotated rx -180 ry -65 rz 16.01 deg; joints [2.048, 2.049, 21.877, -54.751, 105.805, -76.306, -2376.008]
  MoveL 1136 to (-49.86, 193.4, 270) mm, rotated rx -180 ry -65 rz 13.18 deg; joints [1.783, 0.938, 24.149, -54.638, 104.939, -75.468, -2373.179]
  MoveL 1137 to (-53.49, 196.56, 260) mm, rotated rx -180 ry -65 rz 9.86 deg; joints [1.518, -0.013, 26.092, -54.579, 104.168, -74.775, -2369.865]
  MoveL 1138 to (-57.36, 200.4, 250) mm, rotated rx 180 ry -65 rz 6.1 deg; joints [1.252, -0.857, 27.817, -54.555, 103.464, -74.178, -2366.095]
  MoveL 1139 to (-62, 207.76, 238.93) mm, rotated rx -180 ry -65 rz 11.9 deg; joints [0.699, 8.07, 10.028, -57.855, 103.914, -73.276, -2361.899]
  MoveL 1140 to (-65.27, 210.27, 230) mm, rotated rx -180 ry -65 rz 7.3 deg; joints [0.435, 6.602, 13.007, -57.668, 102.896, -72.1, -2357.303]
  MoveL 1141 to (-68.98, 216.33, 220) mm, rotated rx -180 ry -65 rz 2.34 deg; joints [0.169, 4.078, 18.116, -57.324, 101.298, -70.007, -2352.338]
  MoveL 1142 to (-72.31, 223.11, 210) mm, rotated rx -180 ry -65 rz -2.97 deg; joints [-0.097, 2.624, 21.059, -57.214, 100.286, -68.866, -2347.029]
  MoveL 1143 to (-75.1, 230.56, 200) mm, rotated rx -180 ry -65 rz -8.6 deg; joints [-0.364, 1.488, 23.357, -57.177, 99.452, -68.009, -2341.404]
  MoveL 1144 to (-77.2, 238.6, 190) mm, rotated rx -180 ry -65 rz -14.51 deg; joints [-0.632, 0.524, 25.303, -57.181, 98.716, -67.306, -2335.49]
  MoveL 1145 to (-78.47, 247.13, 180) mm, rotated rx 180 ry -65 rz -20.68 deg; joints [-0.9, -0.326, 27.017, -57.212, 98.046, -66.704, -2329.316]
  MoveL 1146 to (-76.55, 260.68, 168.28) mm, rotated rx -180 ry -65 rz -17.09 deg; joints [-1.435, 8.019, 10.028, -60.241, 98.247, -65.608, -2322.909]
  MoveL 1147 to (-77.05, 266.7, 159.36) mm, rotated rx -180 ry -65 rz -23.7 deg; joints [-1.702, 8.015, 10.028, -60.342, 98.028, -65.739, -2316.299]
  MoveL 1148 to (-76.31, 274.12, 150) mm, rotated rx -180 ry -65 rz -30.48 deg; joints [-1.97, 10.265, 5.47, -60.739, 98.94, -67.898, -2309.517]
  MoveL 1149 to (-73.44, 283.02, 140) mm, rotated rx 180 ry -65 rz -37.4 deg; joints [-2.239, 12.228, 1.493, -61.116, 99.691, -69.809, -2302.596]
  MoveL 1150 to (-69.5, 291.57, 130) mm, rotated rx -180 ry -65 rz -44.43 deg; joints [-2.508, 13.513, -1.112, -61.401, 100.096, -71.113, -2295.57]
  MoveL 1151 to (-64.57, 299.61, 120) mm, rotated rx -180 ry -65 rz -51.52 deg; joints [-2.779, 14.533, -3.181, -61.646, 100.363, -72.178, -2288.477]
  MoveL 1152 to (-58.74, 306.97, 110) mm, rotated rx -180 ry -65 rz -58.65 deg; joints [-3.051, 15.398, -4.934, -61.865, 100.548, -73.102, -2281.355]
  MoveL 1153 to (-52.14, 313.53, 100) mm, rotated rx 180 ry -65 rz -65.75 deg; joints [-3.324, 16.157, -6.47, -62.065, 100.676, -73.928, -2274.246]
  MoveL 1154 to (-44.91, 319.19, 90) mm, rotated rx -180 ry -65 rz -72.81 deg; joints [-3.597, 16.837, -7.843, -62.25, 100.761, -74.68, -2267.194]
  MoveL 1155 to (-33.66, 324.02, 78.99) mm, rotated rx -180 ry -65 rz -69.76 deg; joints [-4.099, 7.768, 10.028, -63.192, 92.408, -58.156, -2260.242]
  MoveL 1156 to (-28.43, 327.52, 69.76) mm, rotated rx -180 ry -65 rz -76.56 deg; joints [-4.372, 7.772, 10.028, -63.28, 92.175, -58.269, -2253.438]
  MoveL 1157 to (-21.27, 330.31, 60) mm, rotated rx -180 ry -65 rz -83.17 deg; joints [-4.645, 10.428, 4.672, -63.475, 93.15, -60.802, -2246.828]
  MoveL 1158 to (-13.31, 332.11, 50) mm, rotated rx -180 ry -65 rz -89.54 deg; joints [-4.919, 11.934, 1.645, -63.63, 93.59, -62.285, -2240.456]
  MoveL 1159 to (-5.58, 333.04, 40) mm, rotated rx 180 ry -65 rz -95.63 deg; joints [-5.194, 13.002, -0.493, -63.762, 93.824, -63.366, -2234.37]
  MoveL 1160 to (1.77, 333.22, 30) mm, rotated rx -180 ry -65 rz -101.39 deg; joints [-5.47, 13.868, -2.22, -63.881, 93.962, -64.26, -2228.612]
  MoveL 1161 to (8.64, 332.76, 20) mm, rotated rx 180 ry -65 rz -106.77 deg; joints [-5.747, 14.61, -3.694, -63.989, 94.04, -65.038, -2223.227]
  MoveL 1162 to (14.93, 331.81, 10) mm, rotated rx -180 ry -65 rz -111.75 deg; joints [-6.024, 15.266, -4.991, -64.089, 94.075, -65.736, -2218.254]
  MoveL 1163 to (20.57, 330.51, 0) mm, rotated rx -180 ry -65 rz -116.27 deg; joints [-6.302, 15.857, -6.157, -64.183, 94.08, -66.375, -2213.733]
  MoveL 1164 to (-43.85, 188.95, 290) mm, rotated rx -180 ry -65 rz 18.32 deg; joints [2.311, 12.354, 1.025, -57.619, 111.896, -85.415, -2378.321]
  Set speed (60.0 mm/s)
  MoveL 1165 to (-28.22, 202.67, 290) mm, rotated rx 180 ry -65 rz 23.79 deg; joints [2.384, 14.562, -4.643, -58.828, 113.78, -88.566, -2383.793]
  MoveL 1166 to (20.57, 330.51, 0) mm, rotated rx -180 ry -65 rz -116.27 deg; joints [-6.302, 15.857, -6.157, -64.183, 94.08, -66.375, -2213.733]
  Set speed (60.0 mm/s)
  MoveL 1167 to (10.28, 312.41, -0.04) mm, rotated rx -180 ry -65 rz -100.95 deg; joints [-6.444, 6.854, 10.028, -66.338, 87.334, -50.865, -2219.047]
  MoveL 1168 to (20.57, 330.51, 0) mm, rotated rx -180 ry -65 rz -116.27 deg; joints [-6.302, -0.161, 26.213, -64.056, 86.902, -51.671, -2213.733]
  Set speed (60.0 mm/s)
  MoveL 1169 to (14.93, 331.81, 10) mm, rotated rx -180 ry -65 rz -111.75 deg; joints [-6.024, 0.401, 25.047, -63.914, 87.392, -52.104, -2218.254]
  MoveL 1170 to (8.64, 332.76, 20) mm, rotated rx -180 ry -65 rz -106.77 deg; joints [-5.747, 1.03, 23.75, -63.776, 87.913, -52.594, -2223.227]
  MoveL 1171 to (1.77, 333.22, 30) mm, rotated rx -180 ry -65 rz -101.39 deg; joints [-5.47, 1.746, 22.276, -63.644, 88.474, -53.162, -2228.612]
  MoveL 1172 to (-5.58, 333.04, 40) mm, rotated rx -180 ry -65 rz -95.63 deg; joints [-5.194, 2.59, 20.549, -63.519, 89.094, -53.841, -2234.37]
  MoveL 1173 to (-13.31, 332.11, 50) mm, rotated rx 180 ry -65 rz -89.54 deg; joints [-4.919, 3.638, 18.41, -63.405, 89.808, -54.703, -2240.456]
  MoveL 1174 to (-21.27, 330.31, 60) mm, rotated rx -180 ry -65 rz -83.17 deg; joints [-4.645, 5.128, 15.384, -63.311, 90.725, -55.962, -2246.828]
  MoveL 1175 to (-28.43, 327.52, 69.76) mm, rotated rx 180 ry -65 rz -76.56 deg; joints [-4.372, 7.772, 10.028, -63.28, 92.175, -58.269, -2253.438]
  MoveL 1176 to (-33.66, 324.02, 78.99) mm, rotated rx -180 ry -65 rz -69.76 deg; joints [-4.099, 7.768, 10.028, -63.192, 92.408, -58.156, -2260.242]
  MoveL 1177 to (-44.91, 319.19, 90) mm, rotated rx 180 ry -65 rz -72.81 deg; joints [-3.597, -0.849, 27.899, -60.456, 92.048, -58.75, -2267.194]
  MoveL 1178 to (-52.14, 313.53, 100) mm, rotated rx 180 ry -65 rz -65.75 deg; joints [-3.324, -0.17, 26.526, -60.353, 92.604, -59.233, -2274.246]
  MoveL 1179 to (-58.74, 306.97, 110) mm, rotated rx -180 ry -65 rz -58.65 deg; joints [-3.051, 0.591, 24.99, -60.261, 93.201, -59.785, -2281.355]
  MoveL 1180 to (-64.57, 299.61, 120) mm, rotated rx -180 ry -65 rz -51.52 deg; joints [-2.779, 1.461, 23.237, -60.185, 93.853, -60.431, -2288.477]
  MoveL 1181 to (-69.5, 291.57, 130) mm, rotated rx 180 ry -65 rz -44.43 deg; joints [-2.508, 2.488, 21.168, -60.132, 94.585, -61.214, -2295.57]
  MoveL 1182 to (-73.44, 283.02, 140) mm, rotated rx -180 ry -65 rz -37.4 deg; joints [-2.239, 3.782, 18.562, -60.116, 95.454, -62.232, -2302.596]
  MoveL 1183 to (-76.31, 274.12, 150) mm, rotated rx 180 ry -65 rz -30.48 deg; joints [-1.97, 5.754, 14.586, -60.189, 96.669, -63.854, -2309.517]
  MoveL 1184 to (-77.05, 266.7, 159.36) mm, rotated rx -180 ry -65 rz -23.7 deg; joints [-1.702, 8.015, 10.028, -60.342, 98.028, -65.739, -2316.299]
  MoveL 1185 to (-76.55, 260.68, 168.28) mm, rotated rx -180 ry -65 rz -17.09 deg; joints [-1.435, 8.019, 10.028, -60.241, 98.247, -65.608, -2322.909]
  MoveL 1186 to (-78.47, 247.13, 180) mm, rotated rx -180 ry -65 rz -20.68 deg; joints [-0.9, -0.326, 27.017, -57.212, 98.046, -66.704, -2329.316]
  MoveL 1187 to (-77.2, 238.6, 190) mm, rotated rx 180 ry -65 rz -14.51 deg; joints [-0.632, 0.524, 25.303, -57.181, 98.716, -67.306, -2335.49]
  MoveL 1188 to (-75.1, 230.56, 200) mm, rotated rx -180 ry -65 rz -8.6 deg; joints [-0.364, 1.488, 23.357, -57.177, 99.452, -68.009, -2341.404]
  MoveL 1189 to (-72.31, 223.11, 210) mm, rotated rx -180 ry -65 rz -2.97 deg; joints [-0.097, 2.624, 21.059, -57.214, 100.286, -68.866, -2347.029]
  MoveL 1190 to (-68.98, 216.33, 220) mm, rotated rx -180 ry -65 rz 2.34 deg; joints [0.169, 4.078, 18.116, -57.324, 101.298, -70.007, -2352.338]
  MoveL 1191 to (-65.27, 210.27, 230) mm, rotated rx -180 ry -65 rz 7.3 deg; joints [0.435, 6.602, 13.007, -57.668, 102.896, -72.1, -2357.303]
  MoveL 1192 to (-62, 207.76, 238.93) mm, rotated rx 180 ry -65 rz 11.9 deg; joints [0.699, 8.07, 10.028, -57.855, 103.914, -73.276, -2361.899]
  MoveL 1193 to (-57.36, 200.4, 250) mm, rotated rx -180 ry -65 rz 6.1 deg; joints [1.252, -0.857, 27.817, -54.555, 103.464, -74.178, -2366.095]
  MoveL 1194 to (-53.49, 196.56, 260) mm, rotated rx -180 ry -65 rz 9.86 deg; joints [1.518, -0.013, 26.092, -54.579, 104.168, -74.775, -2369.865]
  MoveL 1195 to (-49.86, 193.4, 270) mm, rotated rx -180 ry -65 rz 13.18 deg; joints [1.783, 0.938, 24.149, -54.638, 104.939, -75.468, -2373.179]
  MoveL 1196 to (-46.6, 190.89, 280) mm, rotated rx 180 ry -65 rz 16.01 deg; joints [2.048, 2.049, 21.877, -54.751, 105.805, -76.306, -2376.008]
  MoveL 1197 to (-43.85, 188.95, 290) mm, rotated rx -180 ry -65 rz 18.32 deg; joints [2.311, 3.444, 19.031, -54.954, 106.839, -77.397, -2378.321]
  MoveL 1198 to (-28.22, 202.67, 290) mm, rotated rx -180 ry -65 rz 23.79 deg; joints [2.384, 0.043, 24.698, -54.376, 105.583, -75.432, -2383.793]
  Set speed (60.0 mm/s)
  MoveL 1199 to (-30.4, 203.93, 280) mm, rotated rx -180 ry -65 rz 21.53 deg; joints [2.12, -0.887, 26.604, -54.311, 104.819, -74.754, -2381.533]
  MoveL 1200 to (-35.6, 209.96, 268.01) mm, rotated rx 180 ry -65 rz 28.77 deg; joints [1.558, 7.454, 10.028, -57.615, 104.934, -73.363, -2378.768]
  MoveL 1201 to (-36.68, 209.15, 259.36) mm, rotated rx -180 ry -65 rz 25.53 deg; joints [1.295, 7.465, 10.028, -57.727, 104.716, -73.493, -2375.528]
  MoveL 1202 to (-39.07, 210.28, 250) mm, rotated rx 180 ry -65 rz 21.84 deg; joints [1.031, 4.769, 15.494, -57.269, 103.017, -71.225, -2371.841]
  MoveL 1203 to (-42.34, 213.41, 240) mm, rotated rx -180 ry -65 rz 17.73 deg; joints [0.766, 2.865, 19.356, -57.033, 101.747, -69.677, -2367.735]
  MoveL 1204 to (-45.62, 217.1, 230) mm, rotated rx 180 ry -65 rz 13.24 deg; joints [0.501, 1.552, 22.023, -56.936, 100.805, -68.656, -2363.236]
  MoveL 1205 to (-48.8, 221.36, 220) mm, rotated rx -180 ry -65 rz 8.37 deg; joints [0.235, 0.485, 24.187, -56.901, 100.002, -67.856, -2358.371]
  MoveL 1206 to (-51.74, 226.19, 210) mm, rotated rx -180 ry -65 rz 3.16 deg; joints [-0.032, -0.436, 26.053, -56.902, 99.284, -67.187, -2353.164]
  MoveL 1207 to (-54.33, 231.55, 200) mm, rotated rx -180 ry -65 rz -2.36 deg; joints [-0.3, -1.259, 27.716, -56.929, 98.623, -66.607, -2347.64]
  MoveL 1208 to (-56.06, 240.96, 188.77) mm, rotated rx -180 ry -65 rz 1.82 deg; joints [-0.842, 7.444, 10.028, -60.093, 99.023, -65.828, -2341.825]
  MoveL 1209 to (-57.9, 243.94, 179.9) mm, rotated rx -180 ry -65 rz -4.26 deg; joints [-1.108, 7.441, 10.028, -60.193, 98.804, -65.959, -2335.742]
  MoveL 1210 to (-58.8, 250.25, 170) mm, rotated rx -180 ry -65 rz -10.58 deg; joints [-1.375, 3.96, 17.054, -59.877, 96.815, -62.987, -2329.418]
  MoveL 1211 to (-58.89, 257.04, 160) mm, rotated rx -180 ry -65 rz -17.12 deg; joints [-1.643, 2.411, 20.173, -59.84, 95.811, -61.746, -2322.877]
  MoveL 1212 to (-58.18, 263.92, 150) mm, rotated rx -180 ry -65 rz -23.85 deg; joints [-1.911, 1.246, 22.515, -59.862, 95.006, -60.848, -2316.149]
  MoveL 1213 to (-56.65, 270.74, 140) mm, rotated rx -180 ry -65 rz -30.74 deg; joints [-2.181, 0.277, 24.46, -59.914, 94.304, -60.125, -2309.263]
  MoveL 1214 to (-54.3, 277.38, 130) mm, rotated rx 180 ry -65 rz -37.75 deg; joints [-2.452, -0.566, 26.151, -59.986, 93.667, -59.512, -2302.251]
  MoveL 1215 to (-51.17, 283.7, 120) mm, rotated rx -180 ry -65 rz -44.85 deg; joints [-2.723, -1.316, 27.656, -60.073, 93.079, -58.979, -2295.149]
  MoveL 1216 to (-44.05, 291.51, 108.86) mm, rotated rx -180 ry -65 rz -42.01 deg; joints [-3.234, 7.183, 10.028, -62.94, 93.409, -58.304, -2287.994]
  MoveL 1217 to (-42.07, 295.25, 99.75) mm, rotated rx -180 ry -65 rz -49.17 deg; joints [-3.504, 7.179, 10.028, -63.026, 93.181, -58.425, -2280.828]
  MoveL 1218 to (-37.86, 299.62, 90) mm, rotated rx -180 ry -65 rz -56.3 deg; joints [-3.775, 10.02, 4.283, -63.276, 94.26, -61.14, -2273.695]
  MoveL 1219 to (-32.46, 303.64, 80) mm, rotated rx 180 ry -65 rz -63.36 deg; joints [-4.047, 11.569, 1.151, -63.46, 94.733, -62.678, -2266.643]
  MoveL 1220 to (-26.8, 306.94, 70) mm, rotated rx 180 ry -65 rz -70.28 deg; joints [-4.32, 12.674, -1.081, -63.614, 94.996, -63.809, -2259.72]
  MoveL 1221 to (-21, 309.52, 60) mm, rotated rx -180 ry -65 rz -77.02 deg; joints [-4.594, 13.572, -2.888, -63.75, 95.158, -64.747, -2252.977]
  MoveL 1222 to (-15.19, 311.39, 50) mm, rotated rx -180 ry -65 rz -83.54 deg; joints [-4.869, 14.341, -4.431, -63.873, 95.257, -65.565, -2246.464]
  MoveL 1223 to (-9.5, 312.61, 40) mm, rotated rx 180 ry -65 rz -89.77 deg; joints [-5.145, 15.019, -5.788, -63.986, 95.311, -66.296, -2240.231]
  MoveL 1224 to (-4.03, 313.25, 30) mm, rotated rx -180 ry -65 rz -95.67 deg; joints [-5.421, 15.63, -7.003, -64.091, 95.33, -66.963, -2234.327]
  MoveL 1225 to (5.28, 311.14, 18.82) mm, rotated rx 180 ry -65 rz -91.2 deg; joints [-5.894, 6.832, 10.028, -66.187, 87.825, -50.673, -2228.799]
  MoveL 1226 to (7.88, 311.77, 9.41) mm, rotated rx -180 ry -65 rz -96.31 deg; joints [-6.169, 6.842, 10.028, -66.263, 87.58, -50.77, -2223.692]
  MoveL 1227 to (10.28, 312.41, -0.04) mm, rotated rx -180 ry -65 rz -100.95 deg; joints [-6.444, 6.854, 10.028, -66.338, 87.334, -50.865, -2219.047]
  Set speed (1000.0 mm/s)
  MoveL 1228 to (10.28, 312.41, -0.04) mm, rotated rx -180 ry -65 rz -100.95 deg; joints [-6.444, 6.854, 10.028, -66.338, 87.334, -50.865, -2219.047]
  MoveL 1229 to (12.08, 311, 9.4) mm, rotated rx -180 ry -65 rz -100.95 deg; joints [-6.169, 6.844, 10.028, -66.263, 87.579, -50.768, -2219.047]
